    MoveL RelTool(pTarget,0,0,-2),vSpeed,z0,tTool\WObj:=wWobj;
    MoveL pTarget,vSpeed,fine,tTool\WObj:=wWobj;
    Set do_pen;
    MoveL pTarget,vSpeed,z0,tTool\WObj:=wWobj;
    MoveL pTarget,vSpeed,z0,tTool\WObj:=wWobj;
    MoveL pTarget,vSpeed,z0,tTool\WObj:=wWobj;
    MoveL pTarget,vSpeed,z0,tTool\WObj:=wWobj;
    MoveL pTarget,vSpeed,z0,tTool\WObj:=wWobj;
    MoveL pTarget,vSpeed,z0,tTool\WObj:=wWobj;
    MoveL pTarget,vSpeed,z0,tTool\WObj:=wWobj;
    MoveL pTarget,vSpeed,z0,tTool\WObj:=wWobj;
    MoveL pTarget,vSpeed,fine,tTool\WObj:=wWobj;
    Reset do_pen;
    MoveL RelTool(pTarget,0,0,-2),vSpeed,z0,tTool\WObj:=wWobj;
  ENDPROC
  PROC char_pipe()
    MoveL pTarget,vSpeed,fine,tTool\WObj:=wWobj;
    Set do_pen;
    MoveL pTarget,vSpeed,fine,tTool\WObj:=wWobj;
    Reset do_pen;
    MoveL RelTool(pTarget,0,0,-2),vSpeed,z0,tTool\WObj:=wWobj;
  ENDPROC
  PROC char_lessthan()
    MoveL pTarget,vSpeed,fine,tTool\WObj:=wWobj;
    Set do_pen;
    MoveL pTarget,vSpeed,z0,tTool\WObj:=wWobj;
    MoveL pTarget,vSpeed,fine,tTool\WObj:=wWobj;
    Reset do_pen;
    MoveL RelTool(pTarget,0,0,-2),vSpeed,z0,tTool\WObj:=wWobj;
  ENDPROC
  PROC char_greaterthan()
    MoveL pTarget,vSpeed,fine,tTool\WObj:=wWobj;
    Set do_pen;
    MoveL pTarget,vSpeed,z0,tTool\WObj:=wWobj;
    MoveL pTarget,vSpeed,fine,tTool\WObj:=wWobj;
    Reset do_pen;
    MoveL RelTool(pTarget,0,0,-2),vSpeed,z0,tTool\WObj:=wWobj;
  ENDPROC
  PROC char_question()
    MoveL pTarget,vSpeed,fine,tTool\WObj:=wWobj;
    Set do_pen;
    MoveL pTarget,vSpeed,z0,tTool\WObj:=wWobj;
    MoveL pTarget,vSpeed,z0,tTool\WObj:=wWobj;
    MoveL pTarget,vSpeed,z0,tTool\WObj:=wWobj;
    MoveL pTarget,vSpeed,z0,tTool\WObj:=wWobj;
    MoveL pTarget,vSpeed,z0,tTool\WObj:=wWobj;
    MoveL pTarget,vSpeed,z0,tTool\WObj:=wWobj;
    MoveL pTarget,vSpeed,z0,tTool\WObj:=wWobj;
    MoveL pTarget,vSpeed,z0,tTool\WObj:=wWobj;
    MoveL pTarget,vSpeed,z0,tTool\WObj:=wWobj;
    MoveL pTarget,vSpeed,z0,tTool\WObj:=wWobj;
    MoveL pTarget,vSpeed,z0,tTool\WObj:=wWobj;
    MoveL pTarget,vSpeed,z0,tTool\WObj:=wWobj;
    MoveL pTarget,vSpeed,fine,tTool\WObj:=wWobj;
    Reset do_pen;
    MoveL RelTool(pTarget,0,0,-2),vSpeed,z0,tTool\WObj:=wWobj;
    MoveL pTarget,vSpeed,fine,tTool\WObj:=wWobj;
    Set do_pen;
    MoveL pTarget,vSpeed,z0,tTool\WObj:=wWobj;
    MoveL pTarget,vSpeed,z0,tTool\WObj:=wWobj;
    MoveL pTarget,vSpeed,z0,tTool\WObj:=wWobj;
    MoveL pTarget,vSpeed,fine,tTool\WObj:=wWobj;
    Reset do_pen;
    MoveL RelTool(pTarget,0,0,-2),vSpeed,z0,tTool\WObj:=wWobj;
  ENDPROC
  PROC char_underscore()
    MoveL pTarget,vSpeed,fine,tTool\WObj:=wWobj;
    Set do_pen;
    MoveL pTarget,vSpeed,fine,tTool\WObj:=wWobj;
    Reset do_pen;
    MoveL RelTool(pTarget,0,0,-2),vSpeed,z0,tTool\WObj:=wWobj;
  ENDPROC
  PROC char_minus()
    MoveL pTarget,vSpeed,fine,tTool\WObj:=wWobj;
    Set do_pen;
    MoveL pTarget,vSpeed,fine,tTool\WObj:=wWobj;
    Reset do_pen;
    MoveL RelTool(pTarget,0,0,-2),vSpeed,z0,tTool\WObj:=wWobj;
  ENDPROC
  PROC char_tilde()
    MoveL pTarget,vSpeed,fine,tTool\WObj:=wWobj;
    Set do_pen;
    MoveL pTarget,vSpeed,z0,tTool\WObj:=wWobj;
    MoveL pTarget,vSpeed,z0,tTool\WObj:=wWobj;
    MoveL pTarget,vSpeed,z0,tTool\WObj:=wWobj;
    MoveL pTarget,vSpeed,z0,tTool\WObj:=wWobj;
    MoveL pTarget,vSpeed,z0,tTool\WObj:=wWobj;
    MoveL pTarget,vSpeed,z0,tTool\WObj:=wWobj;
    MoveL pTarget,vSpeed,z0,tTool\WObj:=wWobj;
    MoveL pTarget,vSpeed,z0,tTool\WObj:=wWobj;
    MoveL pTarget,vSpeed,z0,tTool\WObj:=wWobj;
    MoveL pTarget,vSpeed,fine,tTool\WObj:=wWobj;
    Reset do_pen;
    MoveL RelTool(pTarget,0,0,-2),vSpeed,z0,tTool\WObj:=wWobj;
    MoveL pTarget,vSpeed,fine,tTool\WObj:=wWobj;
    Set do_pen;
    MoveL pTarget,vSpeed,z0,tTool\WObj:=wWobj;
    MoveL pTarget,vSpeed,z0,tTool\WObj:=wWobj;
    MoveL pTarget,vSpeed,z0,tTool\WObj:=wWobj;
    MoveL pTarget,vSpeed,z0,tTool\WObj:=wWobj;
    MoveL pTarget,vSpeed,z0,tTool\WObj:=wWobj;
    MoveL pTarget,vSpeed,z0,tTool\WObj:=wWobj;
    MoveL pTarget,vSpeed,z0,tTool\WObj:=wWobj;
    MoveL pTarget,vSpeed,z0,tTool\WObj:=wWobj;
    MoveL pTarget,vSpeed,z0,tTool\WObj:=wWobj;
    MoveL pTarget,vSpeed,fine,tTool\WObj:=wWobj;
    Reset do_pen;
    MoveL RelTool(pTarget,0,0,-2),vSpeed,z0,tTool\WObj:=wWobj;
  ENDPROC
  PROC char_period()
    MoveL pTarget,vSpeed,fine,tTool\WObj:=wWobj;
    Set do_pen;
    MoveL pTarget,vSpeed,z0,tTool\WObj:=wWobj;
    MoveL pTarget,vSpeed,z0,tTool\WObj:=wWobj;
    MoveL pTarget,vSpeed,z0,tTool\WObj:=wWobj;
    MoveL pTarget,vSpeed,fine,tTool\WObj:=wWobj;
    Reset do_pen;
    MoveL RelTool(pTarget,0,0,-2),vSpeed,z0,tTool\WObj:=wWobj;
  ENDPROC
  PROC char_comma()
    MoveL pTarget,vSpeed,fine,tTool\WObj:=wWobj;
    Set do_pen;
    MoveL pTarget,vSpeed,z0,tTool\WObj:=wWobj;
    MoveL pTarget,vSpeed,z0,tTool\WObj:=wWobj;
    MoveL pTarget,vSpeed,z0,tTool\WObj:=wWobj;
    MoveL pTarget,vSpeed,z0,tTool\WObj:=wWobj;
    MoveL pTarget,vSpeed,z0,tTool\WObj:=wWobj;
    MoveL pTarget,vSpeed,fine,tTool\WObj:=wWobj;
    Reset do_pen;
    MoveL RelTool(pTarget,0,0,-2),vSpeed,z0,tTool\WObj:=wWobj;
  ENDPROC
  PROC char_semicolon()
    MoveL pTarget,vSpeed,fine,tTool\WObj:=wWobj;
    Set do_pen;
    MoveL pTarget,vSpeed,z0,tTool\WObj:=wWobj;
    MoveL pTarget,vSpeed,z0,tTool\WObj:=wWobj;
    MoveL pTarget,vSpeed,z0,tTool\WObj:=wWobj;
    MoveL pTarget,vSpeed,fine,tTool\WObj:=wWobj;
    Reset do_pen;
    MoveL RelTool(pTarget,0,0,-2),vSpeed,z0,tTool\WObj:=wWobj;
    MoveL pTarget,vSpeed,fine,tTool\WObj:=wWobj;
    Set do_pen;
    MoveL pTarget,vSpeed,z0,tTool\WObj:=wWobj;
    MoveL pTarget,vSpeed,z0,tTool\WObj:=wWobj;
    MoveL pTarget,vSpeed,z0,tTool\WObj:=wWobj;
    MoveL pTarget,vSpeed,z0,tTool\WObj:=wWobj;
    MoveL pTarget,vSpeed,z0,tTool\WObj:=wWobj;
    MoveL pTarget,vSpeed,fine,tTool\WObj:=wWobj;
    Reset do_pen;
    MoveL RelTool(pTarget,0,0,-2),vSpeed,z0,tTool\WObj:=wWobj;
  ENDPROC
  PROC char_colon()
    MoveL pTarget,vSpeed,fine,tTool\WObj:=wWobj;
    Set do_pen;
    MoveL pTarget,vSpeed,z0,tTool\WObj:=wWobj;
    MoveL pTarget,vSpeed,z0,tTool\WObj:=wWobj;
    MoveL pTarget,vSpeed,z0,tTool\WObj:=wWobj;
    MoveL pTarget,vSpeed,fine,tTool\WObj:=wWobj;
    Reset do_pen;
    MoveL RelTool(pTarget,0,0,-2),vSpeed,z0,tTool\WObj:=wWobj;
    MoveL pTarget,vSpeed,fine,tTool\WObj:=wWobj;
    Set do_pen;
    MoveL pTarget,vSpeed,z0,tTool\WObj:=wWobj;
    MoveL pTarget,vSpeed,z0,tTool\WObj:=wWobj;
    MoveL pTarget,vSpeed,z0,tTool\WObj:=wWobj;
    MoveL pTarget,vSpeed,fine,tTool\WObj:=wWobj;
    Reset do_pen;
    MoveL RelTool(pTarget,0,0,-2),vSpeed,z0,tTool\WObj:=wWobj;
  ENDPROC
ENDMODULE


--- Controller Data/IRB1200_5_90/RAPID/TASK1/PROGMOD/hersheyCursiveModule.modx ---
MODULE hersheyCursiveModule
    ! Character: a
    PROC char_a(\num nScaleParam)
        VAR robtarget pTarget;
        VAR num nScale:=1;
        pTarget:=refTarget;
        IF Present(nScaleParam) THEN
            nScale:=nScaleParam;
        ENDIF
        pTarget.trans:=[9*nScale,17.0*nScale,0];
        MoveL pTarget,vSpeed,fine,tTool\WObj:=wWobj;
        Set do_pen;
        pTarget.trans:=[8*nScale,19.0*nScale,0];
        MoveL pTarget,vSpeed,z0,tTool\WObj:=wWobj;
        pTarget.trans:=[6*nScale,20.0*nScale,0];
        MoveL pTarget,vSpeed,z0,tTool\WObj:=wWobj;
        pTarget.trans:=[4*nScale,20.0*nScale,0];
        MoveL pTarget,vSpeed,z0,tTool\WObj:=wWobj;
        pTarget.trans:=[2*nScale,19.0*nScale,0];
        MoveL pTarget,vSpeed,z0,tTool\WObj:=wWobj;
        pTarget.trans:=[1*nScale,18.0*nScale,0];
        MoveL pTarget,vSpeed,z0,tTool\WObj:=wWobj;
        pTarget.trans:=[0*nScale,16.0*nScale,0];
        MoveL pTarget,vSpeed,z0,tTool\WObj:=wWobj;
        pTarget.trans:=[0*nScale,14.0*nScale,0];
        MoveL pTarget,vSpeed,z0,tTool\WObj:=wWobj;
        pTarget.trans:=[1*nScale,12.0*nScale,0];
        MoveL pTarget,vSpeed,z0,tTool\WObj:=wWobj;
        pTarget.trans:=[3*nScale,11.0*nScale,0];
        MoveL pTarget,vSpeed,z0,tTool\WObj:=wWobj;
        pTarget.trans:=[5*nScale,11.0*nScale,0];
        MoveL pTarget,vSpeed,z0,tTool\WObj:=wWobj;
        pTarget.trans:=[7*nScale,12.0*nScale,0];
        MoveL pTarget,vSpeed,z0,tTool\WObj:=wWobj;
        pTarget.trans:=[8*nScale,14.0*nScale,0];
        MoveL pTarget,vSpeed,z0,tTool\WObj:=wWobj;
        pTarget.trans:=[10*nScale,20.0*nScale,0];
        MoveL pTarget,vSpeed,z0,tTool\WObj:=wWobj;
        pTarget.trans:=[9*nScale,15.0*nScale,0];
        MoveL pTarget,vSpeed,z0,tTool\WObj:=wWobj;
        pTarget.trans:=[9*nScale,12.0*nScale,0];
        MoveL pTarget,vSpeed,z0,tTool\WObj:=wWobj;
        pTarget.trans:=[10*nScale,11.0*nScale,0];
        MoveL pTarget,vSpeed,z0,tTool\WObj:=wWobj;
        pTarget.trans:=[11*nScale,11.0*nScale,0];
        MoveL pTarget,vSpeed,z0,tTool\WObj:=wWobj;
        pTarget.trans:=[13*nScale,12.0*nScale,0];
        MoveL pTarget,vSpeed,z0,tTool\WObj:=wWobj;
        pTarget.trans:=[14*nScale,13.0*nScale,0];
        MoveL pTarget,vSpeed,z0,tTool\WObj:=wWobj;
        pTarget.trans:=[16*nScale,16.0*nScale,0];
        MoveL pTarget,vSpeed,fine,tTool\WObj:=wWobj;
        Reset do_pen;
        MoveL RelTool(pTarget,0,0,-2),vSpeed,z0,tTool\WObj:=wWobj;
        wWobj.oframe.trans.x:=wWobj.oframe.trans.x+16*nScale;
    ENDPROC

    ! Character: b
    PROC char_b(\num nScaleParam)
        VAR robtarget pTarget;
        VAR num nScale:=1;
        pTarget:=refTarget;
        IF Present(nScaleParam) THEN
            nScale:=nScaleParam;
        ENDIF
        pTarget.trans:=[0*nScale,16.0*nScale,0];
        MoveL pTarget,vSpeed,fine,tTool\WObj:=wWobj;
        Set do_pen;
        pTarget.trans:=[2*nScale,19.0*nScale,0];
        MoveL pTarget,vSpeed,z0,tTool\WObj:=wWobj;
        pTarget.trans:=[5*nScale,24.0*nScale,0];
        MoveL pTarget,vSpeed,z0,tTool\WObj:=wWobj;
        pTarget.trans:=[6*nScale,26.0*nScale,0];
        MoveL pTarget,vSpeed,z0,tTool\WObj:=wWobj;
        pTarget.trans:=[7*nScale,29.0*nScale,0];
        MoveL pTarget,vSpeed,z0,tTool\WObj:=wWobj;
        pTarget.trans:=[7*nScale,31.0*nScale,0];
        MoveL pTarget,vSpeed,z0,tTool\WObj:=wWobj;
        pTarget.trans:=[6*nScale,32.0*nScale,0];
        MoveL pTarget,vSpeed,z0,tTool\WObj:=wWobj;
        pTarget.trans:=[4*nScale,31.0*nScale,0];
        MoveL pTarget,vSpeed,z0,tTool\WObj:=wWobj;
        pTarget.trans:=[3*nScale,29.0*nScale,0];
        MoveL pTarget,vSpeed,z0,tTool\WObj:=wWobj;
        pTarget.trans:=[2*nScale,25.0*nScale,0];
        MoveL pTarget,vSpeed,z0,tTool\WObj:=wWobj;
        pTarget.trans:=[1*nScale,18.0*nScale,0];
        MoveL pTarget,vSpeed,z0,tTool\WObj:=wWobj;
        pTarget.trans:=[1*nScale,12.0*nScale,0];
        MoveL pTarget,vSpeed,z0,tTool\WObj:=wWobj;
        pTarget.trans:=[2*nScale,11.0*nScale,0];
        MoveL pTarget,vSpeed,z0,tTool\WObj:=wWobj;
        pTarget.trans:=[3*nScale,11.0*nScale,0];
        MoveL pTarget,vSpeed,z0,tTool\WObj:=wWobj;
        pTarget.trans:=[5*nScale,12.0*nScale,0];
        MoveL pTarget,vSpeed,z0,tTool\WObj:=wWobj;
        pTarget.trans:=[7*nScale,14.0*nScale,0];
        MoveL pTarget,vSpeed,z0,tTool\WObj:=wWobj;
        pTarget.trans:=[8*nScale,17.0*nScale,0];
        MoveL pTarget,vSpeed,z0,tTool\WObj:=wWobj;
        pTarget.trans:=[8*nScale,20.0*nScale,0];
        MoveL pTarget,vSpeed,z0,tTool\WObj:=wWobj;
        pTarget.trans:=[9*nScale,16.0*nScale,0];
        MoveL pTarget,vSpeed,z0,tTool\WObj:=wWobj;
        pTarget.trans:=[10*nScale,15.0*nScale,0];
        MoveL pTarget,vSpeed,z0,tTool\WObj:=wWobj;
        pTarget.trans:=[12*nScale,15.0*nScale,0];
        MoveL pTarget,vSpeed,z0,tTool\WObj:=wWobj;
        pTarget.trans:=[14*nScale,16.0*nScale,0];
        MoveL pTarget,vSpeed,fine,tTool\WObj:=wWobj;
        Reset do_pen;
        MoveL RelTool(pTarget,0,0,-2),vSpeed,z0,tTool\WObj:=wWobj;
        wWobj.oframe.trans.x:=wWobj.oframe.trans.x+14*nScale;
    ENDPROC

    ! Character: c
    PROC char_c(\num nScaleParam)
        VAR robtarget pTarget;
        VAR num nScale:=1;
        pTarget:=refTarget;
        IF Present(nScaleParam) THEN
            nScale:=nScaleParam;
        ENDIF
        pTarget.trans:=[7*nScale,18.0*nScale,0];
        MoveL pTarget,vSpeed,fine,tTool\WObj:=wWobj;
        Set do_pen;
        pTarget.trans:=[7*nScale,19.0*nScale,0];
        MoveL pTarget,vSpeed,z0,tTool\WObj:=wWobj;
        pTarget.trans:=[6*nScale,20.0*nScale,0];
        MoveL pTarget,vSpeed,z0,tTool\WObj:=wWobj;
        pTarget.trans:=[4*nScale,20.0*nScale,0];
        MoveL pTarget,vSpeed,z0,tTool\WObj:=wWobj;
        pTarget.trans:=[2*nScale,19.0*nScale,0];
        MoveL pTarget,vSpeed,z0,tTool\WObj:=wWobj;
        pTarget.trans:=[1*nScale,18.0*nScale,0];
        MoveL pTarget,vSpeed,z0,tTool\WObj:=wWobj;
        pTarget.trans:=[0*nScale,16.0*nScale,0];
        MoveL pTarget,vSpeed,z0,tTool\WObj:=wWobj;
        pTarget.trans:=[0*nScale,14.0*nScale,0];
        MoveL pTarget,vSpeed,z0,tTool\WObj:=wWobj;
        pTarget.trans:=[1*nScale,12.0*nScale,0];
        MoveL pTarget,vSpeed,z0,tTool\WObj:=wWobj;
        pTarget.trans:=[3*nScale,11.0*nScale,0];
        MoveL pTarget,vSpeed,z0,tTool\WObj:=wWobj;
        pTarget.trans:=[6*nScale,11.0*nScale,0];
        MoveL pTarget,vSpeed,z0,tTool\WObj:=wWobj;
        pTarget.trans:=[9*nScale,13.0*nScale,0];
        MoveL pTarget,vSpeed,z0,tTool\WObj:=wWobj;
        pTarget.trans:=[11*nScale,16.0*nScale,0];
        MoveL pTarget,vSpeed,fine,tTool\WObj:=wWobj;
        Reset do_pen;
        MoveL RelTool(pTarget,0,0,-2),vSpeed,z0,tTool\WObj:=wWobj;
        wWobj.oframe.trans.x:=wWobj.oframe.trans.x+11*nScale;
    ENDPROC

    ! Character: d
    PROC char_d(\num nScaleParam)
        VAR robtarget pTarget;
        VAR num nScale:=1;
        pTarget:=refTarget;
        IF Present(nScaleParam) THEN
            nScale:=nScaleParam;
        ENDIF
        pTarget.trans:=[9*nScale,17.0*nScale,0];
        MoveL pTarget,vSpeed,fine,tTool\WObj:=wWobj;
        Set do_pen;
        pTarget.trans:=[8*nScale,19.0*nScale,0];
        MoveL pTarget,vSpeed,z0,tTool\WObj:=wWobj;
        pTarget.trans:=[6*nScale,20.0*nScale,0];
        MoveL pTarget,vSpeed,z0,tTool\WObj:=wWobj;
        pTarget.trans:=[4*nScale,20.0*nScale,0];
        MoveL pTarget,vSpeed,z0,tTool\WObj:=wWobj;
        pTarget.trans:=[2*nScale,19.0*nScale,0];
        MoveL pTarget,vSpeed,z0,tTool\WObj:=wWobj;
        pTarget.trans:=[1*nScale,18.0*nScale,0];
        MoveL pTarget,vSpeed,z0,tTool\WObj:=wWobj;
        pTarget.trans:=[0*nScale,16.0*nScale,0];
        MoveL pTarget,vSpeed,z0,tTool\WObj:=wWobj;
        pTarget.trans:=[0*nScale,14.0*nScale,0];
        MoveL pTarget,vSpeed,z0,tTool\WObj:=wWobj;
        pTarget.trans:=[1*nScale,12.0*nScale,0];
        MoveL pTarget,vSpeed,z0,tTool\WObj:=wWobj;
        pTarget.trans:=[3*nScale,11.0*nScale,0];
        MoveL pTarget,vSpeed,z0,tTool\WObj:=wWobj;
        pTarget.trans:=[5*nScale,11.0*nScale,0];
        MoveL pTarget,vSpeed,z0,tTool\WObj:=wWobj;
        pTarget.trans:=[7*nScale,12.0*nScale,0];
        MoveL pTarget,vSpeed,z0,tTool\WObj:=wWobj;
        pTarget.trans:=[8*nScale,14.0*nScale,0];
        MoveL pTarget,vSpeed,z0,tTool\WObj:=wWobj;
        pTarget.trans:=[14*nScale,32.0*nScale,0];
        MoveL pTarget,vSpeed,fine,tTool\WObj:=wWobj;
        Reset do_pen;
        MoveL RelTool(pTarget,0,0,-2),vSpeed,z0,tTool\WObj:=wWobj;
        pTarget.trans:=[10*nScale,20.0*nScale,0];
        MoveL pTarget,vSpeed,fine,tTool\WObj:=wWobj;
        Set do_pen;
        pTarget.trans:=[9*nScale,15.0*nScale,0];
        MoveL pTarget,vSpeed,z0,tTool\WObj:=wWobj;
        pTarget.trans:=[9*nScale,12.0*nScale,0];
        MoveL pTarget,vSpeed,z0,tTool\WObj:=wWobj;
        pTarget.trans:=[10*nScale,11.0*nScale,0];
        MoveL pTarget,vSpeed,z0,tTool\WObj:=wWobj;
        pTarget.trans:=[11*nScale,11.0*nScale,0];
        MoveL pTarget,vSpeed,z0,tTool\WObj:=wWobj;
        pTarget.trans:=[13*nScale,12.0*nScale,0];
        MoveL pTarget,vSpeed,z0,tTool\WObj:=wWobj;
        pTarget.trans:=[14*nScale,13.0*nScale,0];
        MoveL pTarget,vSpeed,z0,tTool\WObj:=wWobj;
        pTarget.trans:=[16*nScale,16.0*nScale,0];
        MoveL pTarget,vSpeed,fine,tTool\WObj:=wWobj;
        Reset do_pen;
        MoveL RelTool(pTarget,0,0,-2),vSpeed,z0,tTool\WObj:=wWobj;
        wWobj.oframe.trans.x:=wWobj.oframe.trans.x+16*nScale;
    ENDPROC

    ! Character: e
    PROC char_e(\num nScaleParam)
        VAR robtarget pTarget;
        VAR num nScale:=1;
        pTarget:=refTarget;
        IF Present(nScaleParam) THEN
            nScale:=nScaleParam;
        ENDIF
        pTarget.trans:=[1*nScale,13.0*nScale,0];
        MoveL pTarget,vSpeed,fine,tTool\WObj:=wWobj;
        Set do_pen;
        pTarget.trans:=[3*nScale,14.0*nScale,0];
        MoveL pTarget,vSpeed,z0,tTool\WObj:=wWobj;
        pTarget.trans:=[4*nScale,15.0*nScale,0];
        MoveL pTarget,vSpeed,z0,tTool\WObj:=wWobj;
        pTarget.trans:=[5*nScale,17.0*nScale,0];
        MoveL pTarget,vSpeed,z0,tTool\WObj:=wWobj;
        pTarget.trans:=[5*nScale,19.0*nScale,0];
        MoveL pTarget,vSpeed,z0,tTool\WObj:=wWobj;
        pTarget.trans:=[4*nScale,20.0*nScale,0];
        MoveL pTarget,vSpeed,z0,tTool\WObj:=wWobj;
        pTarget.trans:=[3*nScale,20.0*nScale,0];
        MoveL pTarget,vSpeed,z0,tTool\WObj:=wWobj;
        pTarget.trans:=[1*nScale,19.0*nScale,0];
        MoveL pTarget,vSpeed,z0,tTool\WObj:=wWobj;
        pTarget.trans:=[0*nScale,17.0*nScale,0];
        MoveL pTarget,vSpeed,z0,tTool\WObj:=wWobj;
        pTarget.trans:=[0*nScale,14.0*nScale,0];
        MoveL pTarget,vSpeed,z0,tTool\WObj:=wWobj;
        pTarget.trans:=[1*nScale,12.0*nScale,0];
        MoveL pTarget,vSpeed,z0,tTool\WObj:=wWobj;
        pTarget.trans:=[3*nScale,11.0*nScale,0];
        MoveL pTarget,vSpeed,z0,tTool\WObj:=wWobj;
        pTarget.trans:=[5*nScale,11.0*nScale,0];
        MoveL pTarget,vSpeed,z0,tTool\WObj:=wWobj;
        pTarget.trans:=[7*nScale,12.0*nScale,0];
        MoveL pTarget,vSpeed,z0,tTool\WObj:=wWobj;
        pTarget.trans:=[8*nScale,13.0*nScale,0];
        MoveL pTarget,vSpeed,z0,tTool\WObj:=wWobj;
        pTarget.trans:=[10*nScale,16.0*nScale,0];
        MoveL pTarget,vSpeed,fine,tTool\WObj:=wWobj;
        Reset do_pen;
        MoveL RelTool(pTarget,0,0,-2),vSpeed,z0,tTool\WObj:=wWobj;
        wWobj.oframe.trans.x:=wWobj.oframe.trans.x+10*nScale;
    ENDPROC

    ! Character: f
    PROC char_f(\num nScaleParam)
        VAR robtarget pTarget;
        VAR num nScale:=1;
        pTarget:=refTarget;
        IF Present(nScaleParam) THEN
            nScale:=nScaleParam;
        ENDIF
        pTarget.trans:=[0*nScale,16.0*nScale,0];
        MoveL pTarget,vSpeed,fine,tTool\WObj:=wWobj;
        Set do_pen;
        pTarget.trans:=[4*nScale,21.0*nScale,0];
        MoveL pTarget,vSpeed,z0,tTool\WObj:=wWobj;
        pTarget.trans:=[6*nScale,24.0*nScale,0];
        MoveL pTarget,vSpeed,z0,tTool\WObj:=wWobj;
        pTarget.trans:=[7*nScale,26.0*nScale,0];
        MoveL pTarget,vSpeed,z0,tTool\WObj:=wWobj;
        pTarget.trans:=[8*nScale,29.0*nScale,0];
        MoveL pTarget,vSpeed,z0,tTool\WObj:=wWobj;
        pTarget.trans:=[8*nScale,31.0*nScale,0];
        MoveL pTarget,vSpeed,z0,tTool\WObj:=wWobj;
        pTarget.trans:=[7*nScale,32.0*nScale,0];
        MoveL pTarget,vSpeed,z0,tTool\WObj:=wWobj;
        pTarget.trans:=[5*nScale,31.0*nScale,0];
        MoveL pTarget,vSpeed,z0,tTool\WObj:=wWobj;
        pTarget.trans:=[4*nScale,29.0*nScale,0];
        MoveL pTarget,vSpeed,z0,tTool\WObj:=wWobj;
        pTarget.trans:=[2*nScale,21.0*nScale,0];
        MoveL pTarget,vSpeed,z0,tTool\WObj:=wWobj;
        pTarget.trans:=[-1*nScale,12.0*nScale,0];
        MoveL pTarget,vSpeed,z0,tTool\WObj:=wWobj;
        pTarget.trans:=[-4*nScale,5.0*nScale,0];
        MoveL pTarget,vSpeed,z0,tTool\WObj:=wWobj;
        pTarget.trans:=[-5*nScale,2.0*nScale,0];
        MoveL pTarget,vSpeed,z0,tTool\WObj:=wWobj;
        pTarget.trans:=[-5*nScale,0.0*nScale,0];
        MoveL pTarget,vSpeed,z0,tTool\WObj:=wWobj;
        pTarget.trans:=[-4*nScale,-1.0*nScale,0];
        MoveL pTarget,vSpeed,z0,tTool\WObj:=wWobj;
        pTarget.trans:=[-2*nScale,0.0*nScale,0];
        MoveL pTarget,vSpeed,z0,tTool\WObj:=wWobj;
        pTarget.trans:=[-1*nScale,3.0*nScale,0];
        MoveL pTarget,vSpeed,z0,tTool\WObj:=wWobj;
        pTarget.trans:=[0*nScale,12.0*nScale,0];
        MoveL pTarget,vSpeed,z0,tTool\WObj:=wWobj;
        pTarget.trans:=[1*nScale,11.0*nScale,0];
        MoveL pTarget,vSpeed,z0,tTool\WObj:=wWobj;
        pTarget.trans:=[3*nScale,11.0*nScale,0];
        MoveL pTarget,vSpeed,z0,tTool\WObj:=wWobj;
        pTarget.trans:=[5*nScale,12.0*nScale,0];
        MoveL pTarget,vSpeed,z0,tTool\WObj:=wWobj;
        pTarget.trans:=[6*nScale,13.0*nScale,0];
        MoveL pTarget,vSpeed,z0,tTool\WObj:=wWobj;
        pTarget.trans:=[8*nScale,16.0*nScale,0];
        MoveL pTarget,vSpeed,fine,tTool\WObj:=wWobj;
        Reset do_pen;
        MoveL RelTool(pTarget,0,0,-2),vSpeed,z0,tTool\WObj:=wWobj;
        wWobj.oframe.trans.x:=wWobj.oframe.trans.x+8*nScale;
    ENDPROC

    ! Character: g
    PROC char_g(\num nScaleParam)
        VAR robtarget pTarget;
        VAR num nScale:=1;
        pTarget:=refTarget;
        IF Present(nScaleParam) THEN
            nScale:=nScaleParam;
        ENDIF
        pTarget.trans:=[9*nScale,17.0*nScale,0];
        MoveL pTarget,vSpeed,fine,tTool\WObj:=wWobj;
        Set do_pen;
        pTarget.trans:=[8*nScale,19.0*nScale,0];
        MoveL pTarget,vSpeed,z0,tTool\WObj:=wWobj;
        pTarget.trans:=[6*nScale,20.0*nScale,0];
        MoveL pTarget,vSpeed,z0,tTool\WObj:=wWobj;
        pTarget.trans:=[4*nScale,20.0*nScale,0];
        MoveL pTarget,vSpeed,z0,tTool\WObj:=wWobj;
        pTarget.trans:=[2*nScale,19.0*nScale,0];
        MoveL pTarget,vSpeed,z0,tTool\WObj:=wWobj;
        pTarget.trans:=[1*nScale,18.0*nScale,0];
        MoveL pTarget,vSpeed,z0,tTool\WObj:=wWobj;
        pTarget.trans:=[0*nScale,16.0*nScale,0];
        MoveL pTarget,vSpeed,z0,tTool\WObj:=wWobj;
        pTarget.trans:=[0*nScale,14.0*nScale,0];
        MoveL pTarget,vSpeed,z0,tTool\WObj:=wWobj;
        pTarget.trans:=[1*nScale,12.0*nScale,0];
        MoveL pTarget,vSpeed,z0,tTool\WObj:=wWobj;
        pTarget.trans:=[3*nScale,11.0*nScale,0];
        MoveL pTarget,vSpeed,z0,tTool\WObj:=wWobj;
        pTarget.trans:=[5*nScale,11.0*nScale,0];
        MoveL pTarget,vSpeed,z0,tTool\WObj:=wWobj;
        pTarget.trans:=[7*nScale,12.0*nScale,0];
        MoveL pTarget,vSpeed,z0,tTool\WObj:=wWobj;
        pTarget.trans:=[8*nScale,13.0*nScale,0];
        MoveL pTarget,vSpeed,fine,tTool\WObj:=wWobj;
        Reset do_pen;
        MoveL RelTool(pTarget,0,0,-2),vSpeed,z0,tTool\WObj:=wWobj;
        pTarget.trans:=[10*nScale,20.0*nScale,0];
        MoveL pTarget,vSpeed,fine,tTool\WObj:=wWobj;
        Set do_pen;
        pTarget.trans:=[8*nScale,13.0*nScale,0];
        MoveL pTarget,vSpeed,z0,tTool\WObj:=wWobj;
        pTarget.trans:=[4*nScale,2.0*nScale,0];
        MoveL pTarget,vSpeed,z0,tTool\WObj:=wWobj;
        pTarget.trans:=[3*nScale,0.0*nScale,0];
        MoveL pTarget,vSpeed,z0,tTool\WObj:=wWobj;
        pTarget.trans:=[1*nScale,-1.0*nScale,0];
        MoveL pTarget,vSpeed,z0,tTool\WObj:=wWobj;
        pTarget.trans:=[0*nScale,0.0*nScale,0];
        MoveL pTarget,vSpeed,z0,tTool\WObj:=wWobj;
        pTarget.trans:=[0*nScale,2.0*nScale,0];
        MoveL pTarget,vSpeed,z0,tTool\WObj:=wWobj;
        pTarget.trans:=[1*nScale,5.0*nScale,0];
        MoveL pTarget,vSpeed,z0,tTool\WObj:=wWobj;
        pTarget.trans:=[4*nScale,8.0*nScale,0];
        MoveL pTarget,vSpeed,z0,tTool\WObj:=wWobj;
        pTarget.trans:=[7*nScale,10.0*nScale,0];
        MoveL pTarget,vSpeed,z0,tTool\WObj:=wWobj;
        pTarget.trans:=[9*nScale,11.0*nScale,0];
        MoveL pTarget,vSpeed,z0,tTool\WObj:=wWobj;
        pTarget.trans:=[12*nScale,13.0*nScale,0];
        MoveL pTarget,vSpeed,z0,tTool\WObj:=wWobj;
        pTarget.trans:=[15*nScale,16.0*nScale,0];
        MoveL pTarget,vSpeed,fine,tTool\WObj:=wWobj;
        Reset do_pen;
        MoveL RelTool(pTarget,0,0,-2),vSpeed,z0,tTool\WObj:=wWobj;
        wWobj.oframe.trans.x:=wWobj.oframe.trans.x+15*nScale;
    ENDPROC

    ! Character: h
    PROC char_h(\num nScaleParam)
        VAR robtarget pTarget;
        VAR num nScale:=1;
        pTarget:=refTarget;
        IF Present(nScaleParam) THEN
            nScale:=nScaleParam;
        ENDIF
        pTarget.trans:=[0*nScale,16.0*nScale,0];
        MoveL pTarget,vSpeed,fine,tTool\WObj:=wWobj;
        Set do_pen;
        pTarget.trans:=[2*nScale,19.0*nScale,0];
        MoveL pTarget,vSpeed,z0,tTool\WObj:=wWobj;
        pTarget.trans:=[5*nScale,24.0*nScale,0];
        MoveL pTarget,vSpeed,z0,tTool\WObj:=wWobj;
        pTarget.trans:=[6*nScale,26.0*nScale,0];
        MoveL pTarget,vSpeed,z0,tTool\WObj:=wWobj;
        pTarget.trans:=[7*nScale,29.0*nScale,0];
        MoveL pTarget,vSpeed,z0,tTool\WObj:=wWobj;
        pTarget.trans:=[7*nScale,31.0*nScale,0];
        MoveL pTarget,vSpeed,z0,tTool\WObj:=wWobj;
        pTarget.trans:=[6*nScale,32.0*nScale,0];
        MoveL pTarget,vSpeed,z0,tTool\WObj:=wWobj;
        pTarget.trans:=[4*nScale,31.0*nScale,0];
        MoveL pTarget,vSpeed,z0,tTool\WObj:=wWobj;
        pTarget.trans:=[3*nScale,29.0*nScale,0];
        MoveL pTarget,vSpeed,z0,tTool\WObj:=wWobj;
        pTarget.trans:=[2*nScale,25.0*nScale,0];
        MoveL pTarget,vSpeed,z0,tTool\WObj:=wWobj;
        pTarget.trans:=[1*nScale,19.0*nScale,0];
        MoveL pTarget,vSpeed,z0,tTool\WObj:=wWobj;
        pTarget.trans:=[0*nScale,11.0*nScale,0];
        MoveL pTarget,vSpeed,fine,tTool\WObj:=wWobj;
        Reset do_pen;
        MoveL RelTool(pTarget,0,0,-2),vSpeed,z0,tTool\WObj:=wWobj;
        pTarget.trans:=[0*nScale,11.0*nScale,0];
        MoveL pTarget,vSpeed,fine,tTool\WObj:=wWobj;
        Set do_pen;
        pTarget.trans:=[1*nScale,14.0*nScale,0];
        MoveL pTarget,vSpeed,z0,tTool\WObj:=wWobj;
        pTarget.trans:=[2*nScale,16.0*nScale,0];
        MoveL pTarget,vSpeed,z0,tTool\WObj:=wWobj;
        pTarget.trans:=[4*nScale,19.0*nScale,0];
        MoveL pTarget,vSpeed,z0,tTool\WObj:=wWobj;
        pTarget.trans:=[6*nScale,20.0*nScale,0];
        MoveL pTarget,vSpeed,z0,tTool\WObj:=wWobj;
        pTarget.trans:=[8*nScale,20.0*nScale,0];
        MoveL pTarget,vSpeed,z0,tTool\WObj:=wWobj;
        pTarget.trans:=[9*nScale,19.0*nScale,0];
        MoveL pTarget,vSpeed,z0,tTool\WObj:=wWobj;
        pTarget.trans:=[9*nScale,17.0*nScale,0];
        MoveL pTarget,vSpeed,z0,tTool\WObj:=wWobj;
        pTarget.trans:=[8*nScale,14.0*nScale,0];
        MoveL pTarget,vSpeed,z0,tTool\WObj:=wWobj;
        pTarget.trans:=[8*nScale,12.0*nScale,0];
        MoveL pTarget,vSpeed,z0,tTool\WObj:=wWobj;
        pTarget.trans:=[9*nScale,11.0*nScale,0];
        MoveL pTarget,vSpeed,z0,tTool\WObj:=wWobj;
        pTarget.trans:=[10*nScale,11.0*nScale,0];
        MoveL pTarget,vSpeed,z0,tTool\WObj:=wWobj;
        pTarget.trans:=[12*nScale,12.0*nScale,0];
        MoveL pTarget,vSpeed,z0,tTool\WObj:=wWobj;
        pTarget.trans:=[13*nScale,13.0*nScale,0];
        MoveL pTarget,vSpeed,z0,tTool\WObj:=wWobj;
        pTarget.trans:=[15*nScale,16.0*nScale,0];
        MoveL pTarget,vSpeed,fine,tTool\WObj:=wWobj;
        Reset do_pen;
        MoveL RelTool(pTarget,0,0,-2),vSpeed,z0,tTool\WObj:=wWobj;
        wWobj.oframe.trans.x:=wWobj.oframe.trans.x+15*nScale;
    ENDPROC

    ! Character: i
    PROC char_i(\num nScaleParam)
        VAR robtarget pTarget;
        VAR num nScale:=1;
        pTarget:=refTarget;
        IF Present(nScaleParam) THEN
            nScale:=nScaleParam;
        ENDIF
        pTarget.trans:=[3*nScale,25.0*nScale,0];
        MoveL pTarget,vSpeed,fine,tTool\WObj:=wWobj;
        Set do_pen;
        pTarget.trans:=[3*nScale,24.0*nScale,0];
        MoveL pTarget,vSpeed,z0,tTool\WObj:=wWobj;
        pTarget.trans:=[4*nScale,24.0*nScale,0];
        MoveL pTarget,vSpeed,z0,tTool\WObj:=wWobj;
        pTarget.trans:=[4*nScale,25.0*nScale,0];
        MoveL pTarget,vSpeed,z0,tTool\WObj:=wWobj;
        pTarget.trans:=[3*nScale,25.0*nScale,0];
        MoveL pTarget,vSpeed,fine,tTool\WObj:=wWobj;
        Reset do_pen;
        MoveL RelTool(pTarget,0,0,-2),vSpeed,z0,tTool\WObj:=wWobj;
        pTarget.trans:=[0*nScale,16.0*nScale,0];
        MoveL pTarget,vSpeed,fine,tTool\WObj:=wWobj;
        Set do_pen;
        pTarget.trans:=[2*nScale,20.0*nScale,0];
        MoveL pTarget,vSpeed,z0,tTool\WObj:=wWobj;
        pTarget.trans:=[0*nScale,14.0*nScale,0];
        MoveL pTarget,vSpeed,z0,tTool\WObj:=wWobj;
        pTarget.trans:=[0*nScale,12.0*nScale,0];
        MoveL pTarget,vSpeed,z0,tTool\WObj:=wWobj;
        pTarget.trans:=[1*nScale,11.0*nScale,0];
        MoveL pTarget,vSpeed,z0,tTool\WObj:=wWobj;
        pTarget.trans:=[2*nScale,11.0*nScale,0];
        MoveL pTarget,vSpeed,z0,tTool\WObj:=wWobj;
        pTarget.trans:=[4*nScale,12.0*nScale,0];
        MoveL pTarget,vSpeed,z0,tTool\WObj:=wWobj;
        pTarget.trans:=[5*nScale,13.0*nScale,0];
        MoveL pTarget,vSpeed,z0,tTool\WObj:=wWobj;
        pTarget.trans:=[7*nScale,16.0*nScale,0];
        MoveL pTarget,vSpeed,fine,tTool\WObj:=wWobj;
        Reset do_pen;
        MoveL RelTool(pTarget,0,0,-2),vSpeed,z0,tTool\WObj:=wWobj;
        wWobj.oframe.trans.x:=wWobj.oframe.trans.x+7*nScale;
    ENDPROC

    ! Character: j
    PROC char_j(\num nScaleParam)
        VAR robtarget pTarget;
        VAR num nScale:=1;
        pTarget:=refTarget;
        IF Present(nScaleParam) THEN
            nScale:=nScaleParam;
        ENDIF
        pTarget.trans:=[3*nScale,25.0*nScale,0];
        MoveL pTarget,vSpeed,fine,tTool\WObj:=wWobj;
        Set do_pen;
        pTarget.trans:=[3*nScale,24.0*nScale,0];
        MoveL pTarget,vSpeed,z0,tTool\WObj:=wWobj;
        pTarget.trans:=[4*nScale,24.0*nScale,0];
        MoveL pTarget,vSpeed,z0,tTool\WObj:=wWobj;
        pTarget.trans:=[4*nScale,25.0*nScale,0];
        MoveL pTarget,vSpeed,z0,tTool\WObj:=wWobj;
        pTarget.trans:=[3*nScale,25.0*nScale,0];
        MoveL pTarget,vSpeed,fine,tTool\WObj:=wWobj;
        Reset do_pen;
        MoveL RelTool(pTarget,0,0,-2),vSpeed,z0,tTool\WObj:=wWobj;
        pTarget.trans:=[0*nScale,16.0*nScale,0];
        MoveL pTarget,vSpeed,fine,tTool\WObj:=wWobj;
        Set do_pen;
        pTarget.trans:=[2*nScale,20.0*nScale,0];
        MoveL pTarget,vSpeed,z0,tTool\WObj:=wWobj;
        pTarget.trans:=[-4*nScale,2.0*nScale,0];
        MoveL pTarget,vSpeed,z0,tTool\WObj:=wWobj;
        pTarget.trans:=[-5*nScale,0.0*nScale,0];
        MoveL pTarget,vSpeed,z0,tTool\WObj:=wWobj;
        pTarget.trans:=[-7*nScale,-1.0*nScale,0];
        MoveL pTarget,vSpeed,z0,tTool\WObj:=wWobj;
        pTarget.trans:=[-8*nScale,0.0*nScale,0];
        MoveL pTarget,vSpeed,z0,tTool\WObj:=wWobj;
        pTarget.trans:=[-8*nScale,2.0*nScale,0];
        MoveL pTarget,vSpeed,z0,tTool\WObj:=wWobj;
        pTarget.trans:=[-7*nScale,5.0*nScale,0];
        MoveL pTarget,vSpeed,z0,tTool\WObj:=wWobj;
        pTarget.trans:=[-4*nScale,8.0*nScale,0];
        MoveL pTarget,vSpeed,z0,tTool\WObj:=wWobj;
        pTarget.trans:=[-1*nScale,10.0*nScale,0];
        MoveL pTarget,vSpeed,z0,tTool\WObj:=wWobj;
        pTarget.trans:=[1*nScale,11.0*nScale,0];
        MoveL pTarget,vSpeed,z0,tTool\WObj:=wWobj;
        pTarget.trans:=[4*nScale,13.0*nScale,0];
        MoveL pTarget,vSpeed,z0,tTool\WObj:=wWobj;
        pTarget.trans:=[7*nScale,16.0*nScale,0];
        MoveL pTarget,vSpeed,fine,tTool\WObj:=wWobj;
        Reset do_pen;
        MoveL RelTool(pTarget,0,0,-2),vSpeed,z0,tTool\WObj:=wWobj;
        wWobj.oframe.trans.x:=wWobj.oframe.trans.x+7*nScale;
    ENDPROC

    ! Character: k
    PROC char_k(\num nScaleParam)
        VAR robtarget pTarget;
        VAR num nScale:=1;
        pTarget:=refTarget;
        IF Present(nScaleParam) THEN
            nScale:=nScaleParam;
        ENDIF
        pTarget.trans:=[0*nScale,16.0*nScale,0];
        MoveL pTarget,vSpeed,fine,tTool\WObj:=wWobj;
        Set do_pen;
        pTarget.trans:=[2*nScale,19.0*nScale,0];
        MoveL pTarget,vSpeed,z0,tTool\WObj:=wWobj;
        pTarget.trans:=[5*nScale,24.0*nScale,0];
        MoveL pTarget,vSpeed,z0,tTool\WObj:=wWobj;
        pTarget.trans:=[6*nScale,26.0*nScale,0];
        MoveL pTarget,vSpeed,z0,tTool\WObj:=wWobj;
        pTarget.trans:=[7*nScale,29.0*nScale,0];
        MoveL pTarget,vSpeed,z0,tTool\WObj:=wWobj;
        pTarget.trans:=[7*nScale,31.0*nScale,0];
        MoveL pTarget,vSpeed,z0,tTool\WObj:=wWobj;
        pTarget.trans:=[6*nScale,32.0*nScale,0];
        MoveL pTarget,vSpeed,z0,tTool\WObj:=wWobj;
        pTarget.trans:=[4*nScale,31.0*nScale,0];
        MoveL pTarget,vSpeed,z0,tTool\WObj:=wWobj;
        pTarget.trans:=[3*nScale,29.0*nScale,0];
        MoveL pTarget,vSpeed,z0,tTool\WObj:=wWobj;
        pTarget.trans:=[2*nScale,25.0*nScale,0];
        MoveL pTarget,vSpeed,z0,tTool\WObj:=wWobj;
        pTarget.trans:=[1*nScale,19.0*nScale,0];
        MoveL pTarget,vSpeed,z0,tTool\WObj:=wWobj;
        pTarget.trans:=[0*nScale,11.0*nScale,0];
        MoveL pTarget,vSpeed,fine,tTool\WObj:=wWobj;
        Reset do_pen;
        MoveL RelTool(pTarget,0,0,-2),vSpeed,z0,tTool\WObj:=wWobj;
        pTarget.trans:=[0*nScale,11.0*nScale,0];
        MoveL pTarget,vSpeed,fine,tTool\WObj:=wWobj;
        Set do_pen;
        pTarget.trans:=[1*nScale,14.0*nScale,0];
        MoveL pTarget,vSpeed,z0,tTool\WObj:=wWobj;
        pTarget.trans:=[2*nScale,16.0*nScale,0];
        MoveL pTarget,vSpeed,z0,tTool\WObj:=wWobj;
        pTarget.trans:=[4*nScale,19.0*nScale,0];
        MoveL pTarget,vSpeed,z0,tTool\WObj:=wWobj;
        pTarget.trans:=[6*nScale,20.0*nScale,0];
        MoveL pTarget,vSpeed,z0,tTool\WObj:=wWobj;
        pTarget.trans:=[8*nScale,20.0*nScale,0];
        MoveL pTarget,vSpeed,z0,tTool\WObj:=wWobj;
        pTarget.trans:=[9*nScale,19.0*nScale,0];
        MoveL pTarget,vSpeed,z0,tTool\WObj:=wWobj;
        pTarget.trans:=[9*nScale,17.0*nScale,0];
        MoveL pTarget,vSpeed,z0,tTool\WObj:=wWobj;
        pTarget.trans:=[7*nScale,16.0*nScale,0];
        MoveL pTarget,vSpeed,z0,tTool\WObj:=wWobj;
        pTarget.trans:=[4*nScale,16.0*nScale,0];
        MoveL pTarget,vSpeed,fine,tTool\WObj:=wWobj;
        Reset do_pen;
        MoveL RelTool(pTarget,0,0,-2),vSpeed,z0,tTool\WObj:=wWobj;
        pTarget.trans:=[4*nScale,16.0*nScale,0];
        MoveL pTarget,vSpeed,fine,tTool\WObj:=wWobj;
        Set do_pen;
        pTarget.trans:=[6*nScale,15.0*nScale,0];
        MoveL pTarget,vSpeed,z0,tTool\WObj:=wWobj;
        pTarget.trans:=[7*nScale,12.0*nScale,0];
        MoveL pTarget,vSpeed,z0,tTool\WObj:=wWobj;
        pTarget.trans:=[8*nScale,11.0*nScale,0];
        MoveL pTarget,vSpeed,z0,tTool\WObj:=wWobj;
        pTarget.trans:=[9*nScale,11.0*nScale,0];
        MoveL pTarget,vSpeed,z0,tTool\WObj:=wWobj;
        pTarget.trans:=[11*nScale,12.0*nScale,0];
        MoveL pTarget,vSpeed,z0,tTool\WObj:=wWobj;
        pTarget.trans:=[12*nScale,13.0*nScale,0];
        MoveL pTarget,vSpeed,z0,tTool\WObj:=wWobj;
        pTarget.trans:=[14*nScale,16.0*nScale,0];
        MoveL pTarget,vSpeed,fine,tTool\WObj:=wWobj;
        Reset do_pen;
        MoveL RelTool(pTarget,0,0,-2),vSpeed,z0,tTool\WObj:=wWobj;
        wWobj.oframe.trans.x:=wWobj.oframe.trans.x+14*nScale;
    ENDPROC

    ! Character: l
    PROC char_l(\num nScaleParam)
        VAR robtarget pTarget;
        VAR num nScale:=1;
        pTarget:=refTarget;
        IF Present(nScaleParam) THEN
            nScale:=nScaleParam;
        ENDIF
        pTarget.trans:=[0*nScale,16.0*nScale,0];
        MoveL pTarget,vSpeed,fine,tTool\WObj:=wWobj;
        Set do_pen;
        pTarget.trans:=[2*nScale,19.0*nScale,0];
        MoveL pTarget,vSpeed,z0,tTool\WObj:=wWobj;
        pTarget.trans:=[5*nScale,24.0*nScale,0];
        MoveL pTarget,vSpeed,z0,tTool\WObj:=wWobj;
        pTarget.trans:=[6*nScale,26.0*nScale,0];
        MoveL pTarget,vSpeed,z0,tTool\WObj:=wWobj;
        pTarget.trans:=[7*nScale,29.0*nScale,0];
        MoveL pTarget,vSpeed,z0,tTool\WObj:=wWobj;
        pTarget.trans:=[7*nScale,31.0*nScale,0];
        MoveL pTarget,vSpeed,z0,tTool\WObj:=wWobj;
        pTarget.trans:=[6*nScale,32.0*nScale,0];
        MoveL pTarget,vSpeed,z0,tTool\WObj:=wWobj;
        pTarget.trans:=[4*nScale,31.0*nScale,0];
        MoveL pTarget,vSpeed,z0,tTool\WObj:=wWobj;
        pTarget.trans:=[3*nScale,29.0*nScale,0];
        MoveL pTarget,vSpeed,z0,tTool\WObj:=wWobj;
        pTarget.trans:=[2*nScale,25.0*nScale,0];
        MoveL pTarget,vSpeed,z0,tTool\WObj:=wWobj;
        pTarget.trans:=[1*nScale,18.0*nScale,0];
        MoveL pTarget,vSpeed,z0,tTool\WObj:=wWobj;
        pTarget.trans:=[1*nScale,12.0*nScale,0];
        MoveL pTarget,vSpeed,z0,tTool\WObj:=wWobj;
        pTarget.trans:=[2*nScale,11.0*nScale,0];
        MoveL pTarget,vSpeed,z0,tTool\WObj:=wWobj;
        pTarget.trans:=[3*nScale,11.0*nScale,0];
        MoveL pTarget,vSpeed,z0,tTool\WObj:=wWobj;
        pTarget.trans:=[5*nScale,12.0*nScale,0];
        MoveL pTarget,vSpeed,z0,tTool\WObj:=wWobj;
        pTarget.trans:=[6*nScale,13.0*nScale,0];
        MoveL pTarget,vSpeed,z0,tTool\WObj:=wWobj;
        pTarget.trans:=[8*nScale,16.0*nScale,0];
        MoveL pTarget,vSpeed,fine,tTool\WObj:=wWobj;
        Reset do_pen;
        MoveL RelTool(pTarget,0,0,-2),vSpeed,z0,tTool\WObj:=wWobj;
        wWobj.oframe.trans.x:=wWobj.oframe.trans.x+8*nScale;
    ENDPROC

    ! Character: m
    PROC char_m(\num nScaleParam)
        VAR robtarget pTarget;
        VAR num nScale:=1;
        pTarget:=refTarget;
        IF Present(nScaleParam) THEN
            nScale:=nScaleParam;
        ENDIF
        pTarget.trans:=[0*nScale,16.0*nScale,0];
        MoveL pTarget,vSpeed,fine,tTool\WObj:=wWobj;
        Set do_pen;
        pTarget.trans:=[2*nScale,19.0*nScale,0];
        MoveL pTarget,vSpeed,z0,tTool\WObj:=wWobj;
        pTarget.trans:=[4*nScale,20.0*nScale,0];
        MoveL pTarget,vSpeed,z0,tTool\WObj:=wWobj;
        pTarget.trans:=[5*nScale,19.0*nScale,0];
        MoveL pTarget,vSpeed,z0,tTool\WObj:=wWobj;
        pTarget.trans:=[5*nScale,18.0*nScale,0];
        MoveL pTarget,vSpeed,z0,tTool\WObj:=wWobj;
        pTarget.trans:=[4*nScale,14.0*nScale,0];
        MoveL pTarget,vSpeed,z0,tTool\WObj:=wWobj;
        pTarget.trans:=[3*nScale,11.0*nScale,0];
        MoveL pTarget,vSpeed,fine,tTool\WObj:=wWobj;
        Reset do_pen;
        MoveL RelTool(pTarget,0,0,-2),vSpeed,z0,tTool\WObj:=wWobj;
        pTarget.trans:=[4*nScale,14.0*nScale,0];
        MoveL pTarget,vSpeed,fine,tTool\WObj:=wWobj;
        Set do_pen;
        pTarget.trans:=[5*nScale,16.0*nScale,0];
        MoveL pTarget,vSpeed,z0,tTool\WObj:=wWobj;
        pTarget.trans:=[7*nScale,19.0*nScale,0];
        MoveL pTarget,vSpeed,z0,tTool\WObj:=wWobj;
        pTarget.trans:=[9*nScale,20.0*nScale,0];
        MoveL pTarget,vSpeed,z0,tTool\WObj:=wWobj;
        pTarget.trans:=[11*nScale,20.0*nScale,0];
        MoveL pTarget,vSpeed,z0,tTool\WObj:=wWobj;
        pTarget.trans:=[12*nScale,19.0*nScale,0];
        MoveL pTarget,vSpeed,z0,tTool\WObj:=wWobj;
        pTarget.trans:=[12*nScale,18.0*nScale,0];
        MoveL pTarget,vSpeed,z0,tTool\WObj:=wWobj;
        pTarget.trans:=[11*nScale,14.0*nScale,0];
        MoveL pTarget,vSpeed,z0,tTool\WObj:=wWobj;
        pTarget.trans:=[10*nScale,11.0*nScale,0];
        MoveL pTarget,vSpeed,fine,tTool\WObj:=wWobj;
        Reset do_pen;
        MoveL RelTool(pTarget,0,0,-2),vSpeed,z0,tTool\WObj:=wWobj;
        pTarget.trans:=[11*nScale,14.0*nScale,0];
        MoveL pTarget,vSpeed,fine,tTool\WObj:=wWobj;
        Set do_pen;
        pTarget.trans:=[12*nScale,16.0*nScale,0];
        MoveL pTarget,vSpeed,z0,tTool\WObj:=wWobj;
        pTarget.trans:=[14*nScale,19.0*nScale,0];
        MoveL pTarget,vSpeed,z0,tTool\WObj:=wWobj;
        pTarget.trans:=[16*nScale,20.0*nScale,0];
        MoveL pTarget,vSpeed,z0,tTool\WObj:=wWobj;
        pTarget.trans:=[18*nScale,20.0*nScale,0];
        MoveL pTarget,vSpeed,z0,tTool\WObj:=wWobj;
        pTarget.trans:=[19*nScale,19.0*nScale,0];
        MoveL pTarget,vSpeed,z0,tTool\WObj:=wWobj;
        pTarget.trans:=[19*nScale,17.0*nScale,0];
        MoveL pTarget,vSpeed,z0,tTool\WObj:=wWobj;
        pTarget.trans:=[18*nScale,14.0*nScale,0];
        MoveL pTarget,vSpeed,z0,tTool\WObj:=wWobj;
        pTarget.trans:=[18*nScale,12.0*nScale,0];
        MoveL pTarget,vSpeed,z0,tTool\WObj:=wWobj;
        pTarget.trans:=[19*nScale,11.0*nScale,0];
        MoveL pTarget,vSpeed,z0,tTool\WObj:=wWobj;
        pTarget.trans:=[20*nScale,11.0*nScale,0];
        MoveL pTarget,vSpeed,z0,tTool\WObj:=wWobj;
        pTarget.trans:=[22*nScale,12.0*nScale,0];
        MoveL pTarget,vSpeed,z0,tTool\WObj:=wWobj;
        pTarget.trans:=[23*nScale,13.0*nScale,0];
        MoveL pTarget,vSpeed,z0,tTool\WObj:=wWobj;
        pTarget.trans:=[25*nScale,16.0*nScale,0];
        MoveL pTarget,vSpeed,fine,tTool\WObj:=wWobj;
        Reset do_pen;
        MoveL RelTool(pTarget,0,0,-2),vSpeed,z0,tTool\WObj:=wWobj;
        wWobj.oframe.trans.x:=wWobj.oframe.trans.x+25*nScale;
    ENDPROC

    ! Character: n
    PROC char_n(\num nScaleParam)
        VAR robtarget pTarget;
        VAR num nScale:=1;
        pTarget:=refTarget;
        IF Present(nScaleParam) THEN
            nScale:=nScaleParam;
        ENDIF
        pTarget.trans:=[0*nScale,16.0*nScale,0];
        MoveL pTarget,vSpeed,fine,tTool\WObj:=wWobj;
        Set do_pen;
        pTarget.trans:=[2*nScale,19.0*nScale,0];
        MoveL pTarget,vSpeed,z0,tTool\WObj:=wWobj;
        pTarget.trans:=[4*nScale,20.0*nScale,0];
        MoveL pTarget,vSpeed,z0,tTool\WObj:=wWobj;
        pTarget.trans:=[5*nScale,19.0*nScale,0];
        MoveL pTarget,vSpeed,z0,tTool\WObj:=wWobj;
        pTarget.trans:=[5*nScale,18.0*nScale,0];
        MoveL pTarget,vSpeed,z0,tTool\WObj:=wWobj;
        pTarget.trans:=[4*nScale,14.0*nScale,0];
        MoveL pTarget,vSpeed,z0,tTool\WObj:=wWobj;
        pTarget.trans:=[3*nScale,11.0*nScale,0];
        MoveL pTarget,vSpeed,fine,tTool\WObj:=wWobj;
        Reset do_pen;
        MoveL RelTool(pTarget,0,0,-2),vSpeed,z0,tTool\WObj:=wWobj;
        pTarget.trans:=[4*nScale,14.0*nScale,0];
        MoveL pTarget,vSpeed,fine,tTool\WObj:=wWobj;
        Set do_pen;
        pTarget.trans:=[5*nScale,16.0*nScale,0];
        MoveL pTarget,vSpeed,z0,tTool\WObj:=wWobj;
        pTarget.trans:=[7*nScale,19.0*nScale,0];
        MoveL pTarget,vSpeed,z0,tTool\WObj:=wWobj;
        pTarget.trans:=[9*nScale,20.0*nScale,0];
        MoveL pTarget,vSpeed,z0,tTool\WObj:=wWobj;
        pTarget.trans:=[11*nScale,20.0*nScale,0];
        MoveL pTarget,vSpeed,z0,tTool\WObj:=wWobj;
        pTarget.trans:=[12*nScale,19.0*nScale,0];
        MoveL pTarget,vSpeed,z0,tTool\WObj:=wWobj;
        pTarget.trans:=[12*nScale,17.0*nScale,0];
        MoveL pTarget,vSpeed,z0,tTool\WObj:=wWobj;
        pTarget.trans:=[11*nScale,14.0*nScale,0];
        MoveL pTarget,vSpeed,z0,tTool\WObj:=wWobj;
        pTarget.trans:=[11*nScale,12.0*nScale,0];
        MoveL pTarget,vSpeed,z0,tTool\WObj:=wWobj;
        pTarget.trans:=[12*nScale,11.0*nScale,0];
        MoveL pTarget,vSpeed,z0,tTool\WObj:=wWobj;
        pTarget.trans:=[13*nScale,11.0*nScale,0];
        MoveL pTarget,vSpeed,z0,tTool\WObj:=wWobj;
        pTarget.trans:=[15*nScale,12.0*nScale,0];
        MoveL pTarget,vSpeed,z0,tTool\WObj:=wWobj;
        pTarget.trans:=[16*nScale,13.0*nScale,0];
        MoveL pTarget,vSpeed,z0,tTool\WObj:=wWobj;
        pTarget.trans:=[18*nScale,16.0*nScale,0];
        MoveL pTarget,vSpeed,fine,tTool\WObj:=wWobj;
        Reset do_pen;
        MoveL RelTool(pTarget,0,0,-2),vSpeed,z0,tTool\WObj:=wWobj;
        wWobj.oframe.trans.x:=wWobj.oframe.trans.x+18*nScale;
    ENDPROC

    ! Character: o
    PROC char_o(\num nScaleParam)
        VAR robtarget pTarget;
        VAR num nScale:=1;
        pTarget:=refTarget;
        IF Present(nScaleParam) THEN
            nScale:=nScaleParam;
        ENDIF
        pTarget.trans:=[6*nScale,20.0*nScale,0];
        MoveL pTarget,vSpeed,fine,tTool\WObj:=wWobj;
        Set do_pen;
        pTarget.trans:=[4*nScale,20.0*nScale,0];
        MoveL pTarget,vSpeed,z0,tTool\WObj:=wWobj;
        pTarget.trans:=[2*nScale,19.0*nScale,0];
        MoveL pTarget,vSpeed,z0,tTool\WObj:=wWobj;
        pTarget.trans:=[1*nScale,18.0*nScale,0];
        MoveL pTarget,vSpeed,z0,tTool\WObj:=wWobj;
        pTarget.trans:=[0*nScale,16.0*nScale,0];
        MoveL pTarget,vSpeed,z0,tTool\WObj:=wWobj;
        pTarget.trans:=[0*nScale,14.0*nScale,0];
        MoveL pTarget,vSpeed,z0,tTool\WObj:=wWobj;
        pTarget.trans:=[1*nScale,12.0*nScale,0];
        MoveL pTarget,vSpeed,z0,tTool\WObj:=wWobj;
        pTarget.trans:=[3*nScale,11.0*nScale,0];
        MoveL pTarget,vSpeed,z0,tTool\WObj:=wWobj;
        pTarget.trans:=[5*nScale,11.0*nScale,0];
        MoveL pTarget,vSpeed,z0,tTool\WObj:=wWobj;
        pTarget.trans:=[7*nScale,12.0*nScale,0];
        MoveL pTarget,vSpeed,z0,tTool\WObj:=wWobj;
        pTarget.trans:=[8*nScale,13.0*nScale,0];
        MoveL pTarget,vSpeed,z0,tTool\WObj:=wWobj;
        pTarget.trans:=[9*nScale,15.0*nScale,0];
        MoveL pTarget,vSpeed,z0,tTool\WObj:=wWobj;
        pTarget.trans:=[9*nScale,17.0*nScale,0];
        MoveL pTarget,vSpeed,z0,tTool\WObj:=wWobj;
        pTarget.trans:=[8*nScale,19.0*nScale,0];
        MoveL pTarget,vSpeed,z0,tTool\WObj:=wWobj;
        pTarget.trans:=[6*nScale,20.0*nScale,0];
        MoveL pTarget,vSpeed,z0,tTool\WObj:=wWobj;
        pTarget.trans:=[5*nScale,19.0*nScale,0];
        MoveL pTarget,vSpeed,z0,tTool\WObj:=wWobj;
        pTarget.trans:=[5*nScale,17.0*nScale,0];
        MoveL pTarget,vSpeed,z0,tTool\WObj:=wWobj;
        pTarget.trans:=[6*nScale,15.0*nScale,0];
        MoveL pTarget,vSpeed,z0,tTool\WObj:=wWobj;
        pTarget.trans:=[8*nScale,14.0*nScale,0];
        MoveL pTarget,vSpeed,z0,tTool\WObj:=wWobj;
        pTarget.trans:=[11*nScale,14.0*nScale,0];
        MoveL pTarget,vSpeed,z0,tTool\WObj:=wWobj;
        pTarget.trans:=[13*nScale,15.0*nScale,0];
        MoveL pTarget,vSpeed,z0,tTool\WObj:=wWobj;
        pTarget.trans:=[14*nScale,16.0*nScale,0];
        MoveL pTarget,vSpeed,fine,tTool\WObj:=wWobj;
        Reset do_pen;
        MoveL RelTool(pTarget,0,0,-2),vSpeed,z0,tTool\WObj:=wWobj;
        wWobj.oframe.trans.x:=wWobj.oframe.trans.x+14*nScale;
    ENDPROC

    ! Character: p
    PROC char_p(\num nScaleParam)
        VAR robtarget pTarget;
        VAR num nScale:=1;
        pTarget:=refTarget;
        IF Present(nScaleParam) THEN
            nScale:=nScaleParam;
        ENDIF
        pTarget.trans:=[0*nScale,16.0*nScale,0];
        MoveL pTarget,vSpeed,fine,tTool\WObj:=wWobj;
        Set do_pen;
        pTarget.trans:=[2*nScale,19.0*nScale,0];
        MoveL pTarget,vSpeed,z0,tTool\WObj:=wWobj;
        pTarget.trans:=[3*nScale,21.0*nScale,0];
        MoveL pTarget,vSpeed,z0,tTool\WObj:=wWobj;
        pTarget.trans:=[2*nScale,17.0*nScale,0];
        MoveL pTarget,vSpeed,z0,tTool\WObj:=wWobj;
        pTarget.trans:=[-4*nScale,-1.0*nScale,0];
        MoveL pTarget,vSpeed,fine,tTool\WObj:=wWobj;
        Reset do_pen;
        MoveL RelTool(pTarget,0,0,-2),vSpeed,z0,tTool\WObj:=wWobj;
        pTarget.trans:=[2*nScale,17.0*nScale,0];
        MoveL pTarget,vSpeed,fine,tTool\WObj:=wWobj;
        Set do_pen;
        pTarget.trans:=[3*nScale,19.0*nScale,0];
        MoveL pTarget,vSpeed,z0,tTool\WObj:=wWobj;
        pTarget.trans:=[5*nScale,20.0*nScale,0];
        MoveL pTarget,vSpeed,z0,tTool\WObj:=wWobj;
        pTarget.trans:=[7*nScale,20.0*nScale,0];
        MoveL pTarget,vSpeed,z0,tTool\WObj:=wWobj;
        pTarget.trans:=[9*nScale,19.0*nScale,0];
        MoveL pTarget,vSpeed,z0,tTool\WObj:=wWobj;
        pTarget.trans:=[10*nScale,17.0*nScale,0];
        MoveL pTarget,vSpeed,z0,tTool\WObj:=wWobj;
        pTarget.trans:=[10*nScale,15.0*nScale,0];
        MoveL pTarget,vSpeed,z0,tTool\WObj:=wWobj;
        pTarget.trans:=[9*nScale,13.0*nScale,0];
        MoveL pTarget,vSpeed,z0,tTool\WObj:=wWobj;
        pTarget.trans:=[8*nScale,12.0*nScale,0];
        MoveL pTarget,vSpeed,z0,tTool\WObj:=wWobj;
        pTarget.trans:=[6*nScale,11.0*nScale,0];
        MoveL pTarget,vSpeed,fine,tTool\WObj:=wWobj;
        Reset do_pen;
        MoveL RelTool(pTarget,0,0,-2),vSpeed,z0,tTool\WObj:=wWobj;
        pTarget.trans:=[2*nScale,12.0*nScale,0];
        MoveL pTarget,vSpeed,fine,tTool\WObj:=wWobj;
        Set do_pen;
        pTarget.trans:=[4*nScale,11.0*nScale,0];
        MoveL pTarget,vSpeed,z0,tTool\WObj:=wWobj;
        pTarget.trans:=[7*nScale,11.0*nScale,0];
        MoveL pTarget,vSpeed,z0,tTool\WObj:=wWobj;
        pTarget.trans:=[10*nScale,12.0*nScale,0];
        MoveL pTarget,vSpeed,z0,tTool\WObj:=wWobj;
        pTarget.trans:=[12*nScale,13.0*nScale,0];
        MoveL pTarget,vSpeed,z0,tTool\WObj:=wWobj;
        pTarget.trans:=[15*nScale,16.0*nScale,0];
        MoveL pTarget,vSpeed,fine,tTool\WObj:=wWobj;
        Reset do_pen;
        MoveL RelTool(pTarget,0,0,-2),vSpeed,z0,tTool\WObj:=wWobj;
        wWobj.oframe.trans.x:=wWobj.oframe.trans.x+15*nScale;
    ENDPROC

    ! Character: q
    PROC char_q(\num nScaleParam)
        VAR robtarget pTarget;
        VAR num nScale:=1;
        pTarget:=refTarget;
        IF Present(nScaleParam) THEN
            nScale:=nScaleParam;
        ENDIF
        pTarget.trans:=[9*nScale,17.0*nScale,0];
        MoveL pTarget,vSpeed,fine,tTool\WObj:=wWobj;
        Set do_pen;
        pTarget.trans:=[8*nScale,19.0*nScale,0];
        MoveL pTarget,vSpeed,z0,tTool\WObj:=wWobj;
        pTarget.trans:=[6*nScale,20.0*nScale,0];
        MoveL pTarget,vSpeed,z0,tTool\WObj:=wWobj;
        pTarget.trans:=[4*nScale,20.0*nScale,0];
        MoveL pTarget,vSpeed,z0,tTool\WObj:=wWobj;
        pTarget.trans:=[2*nScale,19.0*nScale,0];
        MoveL pTarget,vSpeed,z0,tTool\WObj:=wWobj;
        pTarget.trans:=[1*nScale,18.0*nScale,0];
        MoveL pTarget,vSpeed,z0,tTool\WObj:=wWobj;
        pTarget.trans:=[0*nScale,16.0*nScale,0];
        MoveL pTarget,vSpeed,z0,tTool\WObj:=wWobj;
        pTarget.trans:=[0*nScale,14.0*nScale,0];
        MoveL pTarget,vSpeed,z0,tTool\WObj:=wWobj;
        pTarget.trans:=[1*nScale,12.0*nScale,0];
        MoveL pTarget,vSpeed,z0,tTool\WObj:=wWobj;
        pTarget.trans:=[3*nScale,11.0*nScale,0];
        MoveL pTarget,vSpeed,z0,tTool\WObj:=wWobj;
        pTarget.trans:=[5*nScale,11.0*nScale,0];
        MoveL pTarget,vSpeed,z0,tTool\WObj:=wWobj;
        pTarget.trans:=[7*nScale,12.0*nScale,0];
        MoveL pTarget,vSpeed,fine,tTool\WObj:=wWobj;
        Reset do_pen;
        MoveL RelTool(pTarget,0,0,-2),vSpeed,z0,tTool\WObj:=wWobj;
        pTarget.trans:=[10*nScale,20.0*nScale,0];
        MoveL pTarget,vSpeed,fine,tTool\WObj:=wWobj;
        Set do_pen;
        pTarget.trans:=[9*nScale,17.0*nScale,0];
        MoveL pTarget,vSpeed,z0,tTool\WObj:=wWobj;
        pTarget.trans:=[7*nScale,12.0*nScale,0];
        MoveL pTarget,vSpeed,z0,tTool\WObj:=wWobj;
        pTarget.trans:=[4*nScale,5.0*nScale,0];
        MoveL pTarget,vSpeed,z0,tTool\WObj:=wWobj;
        pTarget.trans:=[3*nScale,2.0*nScale,0];
        MoveL pTarget,vSpeed,z0,tTool\WObj:=wWobj;
        pTarget.trans:=[3*nScale,0.0*nScale,0];
        MoveL pTarget,vSpeed,z0,tTool\WObj:=wWobj;
        pTarget.trans:=[4*nScale,-1.0*nScale,0];
        MoveL pTarget,vSpeed,z0,tTool\WObj:=wWobj;
        pTarget.trans:=[6*nScale,0.0*nScale,0];
        MoveL pTarget,vSpeed,z0,tTool\WObj:=wWobj;
        pTarget.trans:=[7*nScale,3.0*nScale,0];
        MoveL pTarget,vSpeed,z0,tTool\WObj:=wWobj;
        pTarget.trans:=[7*nScale,10.0*nScale,0];
        MoveL pTarget,vSpeed,z0,tTool\WObj:=wWobj;
        pTarget.trans:=[9*nScale,11.0*nScale,0];
        MoveL pTarget,vSpeed,z0,tTool\WObj:=wWobj;
        pTarget.trans:=[12*nScale,13.0*nScale,0];
        MoveL pTarget,vSpeed,z0,tTool\WObj:=wWobj;
        pTarget.trans:=[15*nScale,16.0*nScale,0];
        MoveL pTarget,vSpeed,fine,tTool\WObj:=wWobj;
        Reset do_pen;
        MoveL RelTool(pTarget,0,0,-2),vSpeed,z0,tTool\WObj:=wWobj;
        wWobj.oframe.trans.x:=wWobj.oframe.trans.x+15*nScale;
    ENDPROC

    ! Character: r
    PROC char_r(\num nScaleParam)
        VAR robtarget pTarget;
        VAR num nScale:=1;
        pTarget:=refTarget;
        IF Present(nScaleParam) THEN
            nScale:=nScaleParam;
        ENDIF
        pTarget.trans:=[0*nScale,16.0*nScale,0];
        MoveL pTarget,vSpeed,fine,tTool\WObj:=wWobj;
        Set do_pen;
        pTarget.trans:=[2*nScale,19.0*nScale,0];
        MoveL pTarget,vSpeed,z0,tTool\WObj:=wWobj;
        pTarget.trans:=[3*nScale,21.0*nScale,0];
        MoveL pTarget,vSpeed,z0,tTool\WObj:=wWobj;
        pTarget.trans:=[3*nScale,19.0*nScale,0];
        MoveL pTarget,vSpeed,z0,tTool\WObj:=wWobj;
        pTarget.trans:=[6*nScale,19.0*nScale,0];
        MoveL pTarget,vSpeed,z0,tTool\WObj:=wWobj;
        pTarget.trans:=[7*nScale,18.0*nScale,0];
        MoveL pTarget,vSpeed,z0,tTool\WObj:=wWobj;
        pTarget.trans:=[7*nScale,16.0*nScale,0];
        MoveL pTarget,vSpeed,z0,tTool\WObj:=wWobj;
        pTarget.trans:=[6*nScale,13.0*nScale,0];
        MoveL pTarget,vSpeed,z0,tTool\WObj:=wWobj;
        pTarget.trans:=[6*nScale,12.0*nScale,0];
        MoveL pTarget,vSpeed,z0,tTool\WObj:=wWobj;
        pTarget.trans:=[7*nScale,11.0*nScale,0];
        MoveL pTarget,vSpeed,z0,tTool\WObj:=wWobj;
        pTarget.trans:=[8*nScale,11.0*nScale,0];
        MoveL pTarget,vSpeed,z0,tTool\WObj:=wWobj;
        pTarget.trans:=[10*nScale,12.0*nScale,0];
        MoveL pTarget,vSpeed,z0,tTool\WObj:=wWobj;
        pTarget.trans:=[11*nScale,13.0*nScale,0];
        MoveL pTarget,vSpeed,z0,tTool\WObj:=wWobj;
        pTarget.trans:=[13*nScale,16.0*nScale,0];
        MoveL pTarget,vSpeed,fine,tTool\WObj:=wWobj;
        Reset do_pen;
        MoveL RelTool(pTarget,0,0,-2),vSpeed,z0,tTool\WObj:=wWobj;
        wWobj.oframe.trans.x:=wWobj.oframe.trans.x+13*nScale;
    ENDPROC

    ! Character: s
    PROC char_s(\num nScaleParam)
        VAR robtarget pTarget;
        VAR num nScale:=1;
        pTarget:=refTarget;
        IF Present(nScaleParam) THEN
            nScale:=nScaleParam;
        ENDIF
        pTarget.trans:=[0*nScale,16.0*nScale,0];
        MoveL pTarget,vSpeed,fine,tTool\WObj:=wWobj;
        Set do_pen;
        pTarget.trans:=[2*nScale,19.0*nScale,0];
        MoveL pTarget,vSpeed,z0,tTool\WObj:=wWobj;
        pTarget.trans:=[3*nScale,21.0*nScale,0];
        MoveL pTarget,vSpeed,z0,tTool\WObj:=wWobj;
        pTarget.trans:=[3*nScale,19.0*nScale,0];
        MoveL pTarget,vSpeed,z0,tTool\WObj:=wWobj;
        pTarget.trans:=[5*nScale,16.0*nScale,0];
        MoveL pTarget,vSpeed,z0,tTool\WObj:=wWobj;
        pTarget.trans:=[6*nScale,14.0*nScale,0];
        MoveL pTarget,vSpeed,z0,tTool\WObj:=wWobj;
        pTarget.trans:=[6*nScale,12.0*nScale,0];
        MoveL pTarget,vSpeed,z0,tTool\WObj:=wWobj;
        pTarget.trans:=[4*nScale,11.0*nScale,0];
        MoveL pTarget,vSpeed,fine,tTool\WObj:=wWobj;
        Reset do_pen;
        MoveL RelTool(pTarget,0,0,-2),vSpeed,z0,tTool\WObj:=wWobj;
        pTarget.trans:=[0*nScale,12.0*nScale,0];
        MoveL pTarget,vSpeed,fine,tTool\WObj:=wWobj;
        Set do_pen;
        pTarget.trans:=[2*nScale,11.0*nScale,0];
        MoveL pTarget,vSpeed,z0,tTool\WObj:=wWobj;
        pTarget.trans:=[6*nScale,11.0*nScale,0];
        MoveL pTarget,vSpeed,z0,tTool\WObj:=wWobj;
        pTarget.trans:=[8*nScale,12.0*nScale,0];
        MoveL pTarget,vSpeed,z0,tTool\WObj:=wWobj;
        pTarget.trans:=[9*nScale,13.0*nScale,0];
        MoveL pTarget,vSpeed,z0,tTool\WObj:=wWobj;
        pTarget.trans:=[11*nScale,16.0*nScale,0];
        MoveL pTarget,vSpeed,fine,tTool\WObj:=wWobj;
        Reset do_pen;
        MoveL RelTool(pTarget,0,0,-2),vSpeed,z0,tTool\WObj:=wWobj;
        wWobj.oframe.trans.x:=wWobj.oframe.trans.x+11*nScale;
    ENDPROC

    ! Character: t
    PROC char_t(\num nScaleParam)
        VAR robtarget pTarget;
        VAR num nScale:=1;
        pTarget:=refTarget;
        IF Present(nScaleParam) THEN
            nScale:=nScaleParam;
        ENDIF
        pTarget.trans:=[0*nScale,16.0*nScale,0];
        MoveL pTarget,vSpeed,fine,tTool\WObj:=wWobj;
        Set do_pen;
        pTarget.trans:=[2*nScale,19.0*nScale,0];
        MoveL pTarget,vSpeed,z0,tTool\WObj:=wWobj;
        pTarget.trans:=[4*nScale,23.0*nScale,0];
        MoveL pTarget,vSpeed,fine,tTool\WObj:=wWobj;
        Reset do_pen;
        MoveL RelTool(pTarget,0,0,-2),vSpeed,z0,tTool\WObj:=wWobj;
        pTarget.trans:=[7*nScale,32.0*nScale,0];
        MoveL pTarget,vSpeed,fine,tTool\WObj:=wWobj;
        Set do_pen;
        pTarget.trans:=[1*nScale,14.0*nScale,0];
        MoveL pTarget,vSpeed,z0,tTool\WObj:=wWobj;
        pTarget.trans:=[1*nScale,12.0*nScale,0];
        MoveL pTarget,vSpeed,z0,tTool\WObj:=wWobj;
        pTarget.trans:=[2*nScale,11.0*nScale,0];
        MoveL pTarget,vSpeed,z0,tTool\WObj:=wWobj;
        pTarget.trans:=[4*nScale,11.0*nScale,0];
        MoveL pTarget,vSpeed,z0,tTool\WObj:=wWobj;
        pTarget.trans:=[6*nScale,12.0*nScale,0];
        MoveL pTarget,vSpeed,z0,tTool\WObj:=wWobj;
        pTarget.trans:=[7*nScale,13.0*nScale,0];
        MoveL pTarget,vSpeed,z0,tTool\WObj:=wWobj;
        pTarget.trans:=[9*nScale,16.0*nScale,0];
        MoveL pTarget,vSpeed,fine,tTool\WObj:=wWobj;
        Reset do_pen;
        MoveL RelTool(pTarget,0,0,-2),vSpeed,z0,tTool\WObj:=wWobj;
        pTarget.trans:=[1*nScale,24.0*nScale,0];
        MoveL pTarget,vSpeed,fine,tTool\WObj:=wWobj;
        Set do_pen;
        pTarget.trans:=[8*nScale,24.0*nScale,0];
        MoveL pTarget,vSpeed,fine,tTool\WObj:=wWobj;
        Reset do_pen;
        MoveL RelTool(pTarget,0,0,-2),vSpeed,z0,tTool\WObj:=wWobj;
        wWobj.oframe.trans.x:=wWobj.oframe.trans.x+9*nScale;
    ENDPROC

    ! Character: u
    PROC char_u(\num nScaleParam)
        VAR robtarget pTarget;
        VAR num nScale:=1;
        pTarget:=refTarget;
        IF Present(nScaleParam) THEN
            nScale:=nScaleParam;
        ENDIF
        pTarget.trans:=[0*nScale,16.0*nScale,0];
        MoveL pTarget,vSpeed,fine,tTool\WObj:=wWobj;
        Set do_pen;
        pTarget.trans:=[2*nScale,20.0*nScale,0];
        MoveL pTarget,vSpeed,z0,tTool\WObj:=wWobj;
        pTarget.trans:=[0*nScale,14.0*nScale,0];
        MoveL pTarget,vSpeed,z0,tTool\WObj:=wWobj;
        pTarget.trans:=[0*nScale,12.0*nScale,0];
        MoveL pTarget,vSpeed,z0,tTool\WObj:=wWobj;
        pTarget.trans:=[1*nScale,11.0*nScale,0];
        MoveL pTarget,vSpeed,z0,tTool\WObj:=wWobj;
        pTarget.trans:=[3*nScale,11.0*nScale,0];
        MoveL pTarget,vSpeed,z0,tTool\WObj:=wWobj;
        pTarget.trans:=[5*nScale,12.0*nScale,0];
        MoveL pTarget,vSpeed,z0,tTool\WObj:=wWobj;
        pTarget.trans:=[7*nScale,14.0*nScale,0];
        MoveL pTarget,vSpeed,z0,tTool\WObj:=wWobj;
        pTarget.trans:=[9*nScale,17.0*nScale,0];
        MoveL pTarget,vSpeed,fine,tTool\WObj:=wWobj;
        Reset do_pen;
        MoveL RelTool(pTarget,0,0,-2),vSpeed,z0,tTool\WObj:=wWobj;
        pTarget.trans:=[10*nScale,20.0*nScale,0];
        MoveL pTarget,vSpeed,fine,tTool\WObj:=wWobj;
        Set do_pen;
        pTarget.trans:=[8*nScale,14.0*nScale,0];
        MoveL pTarget,vSpeed,z0,tTool\WObj:=wWobj;
        pTarget.trans:=[8*nScale,12.0*nScale,0];
        MoveL pTarget,vSpeed,z0,tTool\WObj:=wWobj;
        pTarget.trans:=[9*nScale,11.0*nScale,0];
        MoveL pTarget,vSpeed,z0,tTool\WObj:=wWobj;
        pTarget.trans:=[10*nScale,11.0*nScale,0];
        MoveL pTarget,vSpeed,z0,tTool\WObj:=wWobj;
        pTarget.trans:=[12*nScale,12.0*nScale,0];
        MoveL pTarget,vSpeed,z0,tTool\WObj:=wWobj;
        pTarget.trans:=[13*nScale,13.0*nScale,0];
        MoveL pTarget,vSpeed,z0,tTool\WObj:=wWobj;
        pTarget.trans:=[15*nScale,16.0*nScale,0];
        MoveL pTarget,vSpeed,fine,tTool\WObj:=wWobj;
        Reset do_pen;
        MoveL RelTool(pTarget,0,0,-2),vSpeed,z0,tTool\WObj:=wWobj;
        wWobj.oframe.trans.x:=wWobj.oframe.trans.x+15*nScale;
    ENDPROC

    ! Character: v
    PROC char_v(\num nScaleParam)
        VAR robtarget pTarget;
        VAR num nScale:=1;
        pTarget:=refTarget;
        IF Present(nScaleParam) THEN
            nScale:=nScaleParam;
        ENDIF
        pTarget.trans:=[0*nScale,16.0*nScale,0];
        MoveL pTarget,vSpeed,fine,tTool\WObj:=wWobj;
        Set do_pen;
        pTarget.trans:=[2*nScale,20.0*nScale,0];
        MoveL pTarget,vSpeed,z0,tTool\WObj:=wWobj;
        pTarget.trans:=[1*nScale,15.0*nScale,0];
        MoveL pTarget,vSpeed,z0,tTool\WObj:=wWobj;
        pTarget.trans:=[1*nScale,12.0*nScale,0];
        MoveL pTarget,vSpeed,z0,tTool\WObj:=wWobj;
        pTarget.trans:=[2*nScale,11.0*nScale,0];
        MoveL pTarget,vSpeed,z0,tTool\WObj:=wWobj;
        pTarget.trans:=[3*nScale,11.0*nScale,0];
        MoveL pTarget,vSpeed,z0,tTool\WObj:=wWobj;
        pTarget.trans:=[6*nScale,12.0*nScale,0];
        MoveL pTarget,vSpeed,z0,tTool\WObj:=wWobj;
        pTarget.trans:=[8*nScale,14.0*nScale,0];
        MoveL pTarget,vSpeed,z0,tTool\WObj:=wWobj;
        pTarget.trans:=[9*nScale,17.0*nScale,0];
        MoveL pTarget,vSpeed,z0,tTool\WObj:=wWobj;
        pTarget.trans:=[9*nScale,20.0*nScale,0];
        MoveL pTarget,vSpeed,fine,tTool\WObj:=wWobj;
        Reset do_pen;
        MoveL RelTool(pTarget,0,0,-2),vSpeed,z0,tTool\WObj:=wWobj;
        pTarget.trans:=[9*nScale,20.0*nScale,0];
        MoveL pTarget,vSpeed,fine,tTool\WObj:=wWobj;
        Set do_pen;
        pTarget.trans:=[10*nScale,16.0*nScale,0];
        MoveL pTarget,vSpeed,z0,tTool\WObj:=wWobj;
        pTarget.trans:=[11*nScale,15.0*nScale,0];
        MoveL pTarget,vSpeed,z0,tTool\WObj:=wWobj;
        pTarget.trans:=[13*nScale,15.0*nScale,0];
        MoveL pTarget,vSpeed,z0,tTool\WObj:=wWobj;
        pTarget.trans:=[15*nScale,16.0*nScale,0];
        MoveL pTarget,vSpeed,fine,tTool\WObj:=wWobj;
        Reset do_pen;
        MoveL RelTool(pTarget,0,0,-2),vSpeed,z0,tTool\WObj:=wWobj;
        wWobj.oframe.trans.x:=wWobj.oframe.trans.x+15*nScale;
    ENDPROC

    ! Character: w
    PROC char_w(\num nScaleParam)
        VAR robtarget pTarget;
        VAR num nScale:=1;
        pTarget:=refTarget;
        IF Present(nScaleParam) THEN
            nScale:=nScaleParam;
        ENDIF
        pTarget.trans:=[3*nScale,20.0*nScale,0];
        MoveL pTarget,vSpeed,fine,tTool\WObj:=wWobj;
        Set do_pen;
        pTarget.trans:=[1*nScale,18.0*nScale,0];
        MoveL pTarget,vSpeed,z0,tTool\WObj:=wWobj;
        pTarget.trans:=[0*nScale,15.0*nScale,0];
        MoveL pTarget,vSpeed,z0,tTool\WObj:=wWobj;
        pTarget.trans:=[0*nScale,13.0*nScale,0];
        MoveL pTarget,vSpeed,z0,tTool\WObj:=wWobj;
        pTarget.trans:=[1*nScale,11.0*nScale,0];
        MoveL pTarget,vSpeed,z0,tTool\WObj:=wWobj;
        pTarget.trans:=[3*nScale,11.0*nScale,0];
        MoveL pTarget,vSpeed,z0,tTool\WObj:=wWobj;
        pTarget.trans:=[5*nScale,12.0*nScale,0];
        MoveL pTarget,vSpeed,z0,tTool\WObj:=wWobj;
        pTarget.trans:=[7*nScale,14.0*nScale,0];
        MoveL pTarget,vSpeed,fine,tTool\WObj:=wWobj;
        Reset do_pen;
        MoveL RelTool(pTarget,0,0,-2),vSpeed,z0,tTool\WObj:=wWobj;
        pTarget.trans:=[9*nScale,20.0*nScale,0];
        MoveL pTarget,vSpeed,fine,tTool\WObj:=wWobj;
        Set do_pen;
        pTarget.trans:=[7*nScale,14.0*nScale,0];
        MoveL pTarget,vSpeed,z0,tTool\WObj:=wWobj;
        pTarget.trans:=[7*nScale,12.0*nScale,0];
        MoveL pTarget,vSpeed,z0,tTool\WObj:=wWobj;
        pTarget.trans:=[8*nScale,11.0*nScale,0];
        MoveL pTarget,vSpeed,z0,tTool\WObj:=wWobj;
        pTarget.trans:=[10*nScale,11.0*nScale,0];
        MoveL pTarget,vSpeed,z0,tTool\WObj:=wWobj;
        pTarget.trans:=[12*nScale,12.0*nScale,0];
        MoveL pTarget,vSpeed,z0,tTool\WObj:=wWobj;
        pTarget.trans:=[14*nScale,14.0*nScale,0];
        MoveL pTarget,vSpeed,z0,tTool\WObj:=wWobj;
        pTarget.trans:=[15*nScale,17.0*nScale,0];
        MoveL pTarget,vSpeed,z0,tTool\WObj:=wWobj;
        pTarget.trans:=[15*nScale,20.0*nScale,0];
        MoveL pTarget,vSpeed,fine,tTool\WObj:=wWobj;
        Reset do_pen;
        MoveL RelTool(pTarget,0,0,-2),vSpeed,z0,tTool\WObj:=wWobj;
        pTarget.trans:=[15*nScale,20.0*nScale,0];
        MoveL pTarget,vSpeed,fine,tTool\WObj:=wWobj;
        Set do_pen;
        pTarget.trans:=[16*nScale,16.0*nScale,0];
        MoveL pTarget,vSpeed,z0,tTool\WObj:=wWobj;
        pTarget.trans:=[17*nScale,15.0*nScale,0];
        MoveL pTarget,vSpeed,z0,tTool\WObj:=wWobj;
        pTarget.trans:=[19*nScale,15.0*nScale,0];
        MoveL pTarget,vSpeed,z0,tTool\WObj:=wWobj;
        pTarget.trans:=[21*nScale,16.0*nScale,0];
        MoveL pTarget,vSpeed,fine,tTool\WObj:=wWobj;
        Reset do_pen;
        MoveL RelTool(pTarget,0,0,-2),vSpeed,z0,tTool\WObj:=wWobj;
        wWobj.oframe.trans.x:=wWobj.oframe.trans.x+21*nScale;
    ENDPROC

    ! Character: x
    PROC char_x(\num nScaleParam)
        VAR robtarget pTarget;
        VAR num nScale:=1;
        pTarget:=refTarget;
        IF Present(nScaleParam) THEN
            nScale:=nScaleParam;
        ENDIF
        pTarget.trans:=[0*nScale,16.0*nScale,0];
        MoveL pTarget,vSpeed,fine,tTool\WObj:=wWobj;
        Set do_pen;
        pTarget.trans:=[2*nScale,19.0*nScale,0];
        MoveL pTarget,vSpeed,z0,tTool\WObj:=wWobj;
        pTarget.trans:=[4*nScale,20.0*nScale,0];
        MoveL pTarget,vSpeed,z0,tTool\WObj:=wWobj;
        pTarget.trans:=[6*nScale,20.0*nScale,0];
        MoveL pTarget,vSpeed,z0,tTool\WObj:=wWobj;
        pTarget.trans:=[7*nScale,19.0*nScale,0];
        MoveL pTarget,vSpeed,z0,tTool\WObj:=wWobj;
        pTarget.trans:=[7*nScale,12.0*nScale,0];
        MoveL pTarget,vSpeed,z0,tTool\WObj:=wWobj;
        pTarget.trans:=[8*nScale,11.0*nScale,0];
        MoveL pTarget,vSpeed,z0,tTool\WObj:=wWobj;
        pTarget.trans:=[11*nScale,11.0*nScale,0];
        MoveL pTarget,vSpeed,z0,tTool\WObj:=wWobj;
        pTarget.trans:=[14*nScale,13.0*nScale,0];
        MoveL pTarget,vSpeed,z0,tTool\WObj:=wWobj;
        pTarget.trans:=[16*nScale,16.0*nScale,0];
        MoveL pTarget,vSpeed,fine,tTool\WObj:=wWobj;
        Reset do_pen;
        MoveL RelTool(pTarget,0,0,-2),vSpeed,z0,tTool\WObj:=wWobj;
        pTarget.trans:=[13*nScale,19.0*nScale,0];
        MoveL pTarget,vSpeed,fine,tTool\WObj:=wWobj;
        Set do_pen;
        pTarget.trans:=[12*nScale,20.0*nScale,0];
        MoveL pTarget,vSpeed,z0,tTool\WObj:=wWobj;
        pTarget.trans:=[10*nScale,20.0*nScale,0];
        MoveL pTarget,vSpeed,z0,tTool\WObj:=wWobj;
        pTarget.trans:=[9*nScale,19.0*nScale,0];
        MoveL pTarget,vSpeed,z0,tTool\WObj:=wWobj;
        pTarget.trans:=[5*nScale,12.0*nScale,0];
        MoveL pTarget,vSpeed,z0,tTool\WObj:=wWobj;
        pTarget.trans:=[4*nScale,11.0*nScale,0];
        MoveL pTarget,vSpeed,z0,tTool\WObj:=wWobj;
        pTarget.trans:=[2*nScale,11.0*nScale,0];
        MoveL pTarget,vSpeed,z0,tTool\WObj:=wWobj;
        pTarget.trans:=[1*nScale,12.0*nScale,0];
        MoveL pTarget,vSpeed,fine,tTool\WObj:=wWobj;
        Reset do_pen;
        MoveL RelTool(pTarget,0,0,-2),vSpeed,z0,tTool\WObj:=wWobj;
        wWobj.oframe.trans.x:=wWobj.oframe.trans.x+16*nScale;
    ENDPROC

    ! Character: y
    PROC char_y(\num nScaleParam)
        VAR robtarget pTarget;
        VAR num nScale:=1;
        pTarget:=refTarget;
        IF Present(nScaleParam) THEN
            nScale:=nScaleParam;
        ENDIF
        pTarget.trans:=[0*nScale,16.0*nScale,0];
        MoveL pTarget,vSpeed,fine,tTool\WObj:=wWobj;
        Set do_pen;
        pTarget.trans:=[2*nScale,20.0*nScale,0];
        MoveL pTarget,vSpeed,z0,tTool\WObj:=wWobj;
        pTarget.trans:=[0*nScale,14.0*nScale,0];
        MoveL pTarget,vSpeed,z0,tTool\WObj:=wWobj;
        pTarget.trans:=[0*nScale,12.0*nScale,0];
        MoveL pTarget,vSpeed,z0,tTool\WObj:=wWobj;
        pTarget.trans:=[1*nScale,11.0*nScale,0];
        MoveL pTarget,vSpeed,z0,tTool\WObj:=wWobj;
        pTarget.trans:=[3*nScale,11.0*nScale,0];
        MoveL pTarget,vSpeed,z0,tTool\WObj:=wWobj;
        pTarget.trans:=[5*nScale,12.0*nScale,0];
        MoveL pTarget,vSpeed,z0,tTool\WObj:=wWobj;
        pTarget.trans:=[7*nScale,14.0*nScale,0];
        MoveL pTarget,vSpeed,z0,tTool\WObj:=wWobj;
        pTarget.trans:=[9*nScale,17.0*nScale,0];
        MoveL pTarget,vSpeed,fine,tTool\WObj:=wWobj;
        Reset do_pen;
        MoveL RelTool(pTarget,0,0,-2),vSpeed,z0,tTool\WObj:=wWobj;
        pTarget.trans:=[10*nScale,20.0*nScale,0];
        MoveL pTarget,vSpeed,fine,tTool\WObj:=wWobj;
        Set do_pen;
        pTarget.trans:=[4*nScale,2.0*nScale,0];
        MoveL pTarget,vSpeed,z0,tTool\WObj:=wWobj;
        pTarget.trans:=[3*nScale,0.0*nScale,0];
        MoveL pTarget,vSpeed,z0,tTool\WObj:=wWobj;
        pTarget.trans:=[1*nScale,-1.0*nScale,0];
        MoveL pTarget,vSpeed,z0,tTool\WObj:=wWobj;
        pTarget.trans:=[0*nScale,0.0*nScale,0];
        MoveL pTarget,vSpeed,z0,tTool\WObj:=wWobj;
        pTarget.trans:=[0*nScale,2.0*nScale,0];
        MoveL pTarget,vSpeed,z0,tTool\WObj:=wWobj;
        pTarget.trans:=[1*nScale,5.0*nScale,0];
        MoveL pTarget,vSpeed,z0,tTool\WObj:=wWobj;
        pTarget.trans:=[4*nScale,8.0*nScale,0];
        MoveL pTarget,vSpeed,z0,tTool\WObj:=wWobj;
        pTarget.trans:=[7*nScale,10.0*nScale,0];
        MoveL pTarget,vSpeed,z0,tTool\WObj:=wWobj;
        pTarget.trans:=[9*nScale,11.0*nScale,0];
        MoveL pTarget,vSpeed,z0,tTool\WObj:=wWobj;
        pTarget.trans:=[12*nScale,13.0*nScale,0];
        MoveL pTarget,vSpeed,z0,tTool\WObj:=wWobj;
        pTarget.trans:=[15*nScale,16.0*nScale,0];
        MoveL pTarget,vSpeed,fine,tTool\WObj:=wWobj;
        Reset do_pen;
        MoveL RelTool(pTarget,0,0,-2),vSpeed,z0,tTool\WObj:=wWobj;
        wWobj.oframe.trans.x:=wWobj.oframe.trans.x+15*nScale;
    ENDPROC

    ! Character: z
    PROC char_z(\num nScaleParam)
        VAR robtarget pTarget;
        VAR num nScale:=1;
        pTarget:=refTarget;
        IF Present(nScaleParam) THEN
            nScale:=nScaleParam;
        ENDIF
        pTarget.trans:=[0*nScale,16.0*nScale,0];
        MoveL pTarget,vSpeed,fine,tTool\WObj:=wWobj;
        Set do_pen;
        pTarget.trans:=[2*nScale,19.0*nScale,0];
        MoveL pTarget,vSpeed,z0,tTool\WObj:=wWobj;
        pTarget.trans:=[4*nScale,20.0*nScale,0];
        MoveL pTarget,vSpeed,z0,tTool\WObj:=wWobj;
        pTarget.trans:=[6*nScale,20.0*nScale,0];
        MoveL pTarget,vSpeed,z0,tTool\WObj:=wWobj;
        pTarget.trans:=[8*nScale,18.0*nScale,0];
        MoveL pTarget,vSpeed,z0,tTool\WObj:=wWobj;
        pTarget.trans:=[8*nScale,16.0*nScale,0];
        MoveL pTarget,vSpeed,z0,tTool\WObj:=wWobj;
        pTarget.trans:=[7*nScale,14.0*nScale,0];
        MoveL pTarget,vSpeed,z0,tTool\WObj:=wWobj;
        pTarget.trans:=[5*nScale,12.0*nScale,0];
        MoveL pTarget,vSpeed,z0,tTool\WObj:=wWobj;
        pTarget.trans:=[2*nScale,11.0*nScale,0];
        MoveL pTarget,vSpeed,z0,tTool\WObj:=wWobj;
        pTarget.trans:=[4*nScale,10.0*nScale,0];
        MoveL pTarget,vSpeed,z0,tTool\WObj:=wWobj;
        pTarget.trans:=[5*nScale,8.0*nScale,0];
        MoveL pTarget,vSpeed,z0,tTool\WObj:=wWobj;
        pTarget.trans:=[5*nScale,5.0*nScale,0];
        MoveL pTarget,vSpeed,z0,tTool\WObj:=wWobj;
        pTarget.trans:=[4*nScale,2.0*nScale,0];
        MoveL pTarget,vSpeed,z0,tTool\WObj:=wWobj;
        pTarget.trans:=[3*nScale,0.0*nScale,0];
        MoveL pTarget,vSpeed,z0,tTool\WObj:=wWobj;
        pTarget.trans:=[1*nScale,-1.0*nScale,0];
        MoveL pTarget,vSpeed,z0,tTool\WObj:=wWobj;
        pTarget.trans:=[0*nScale,0.0*nScale,0];
        MoveL pTarget,vSpeed,z0,tTool\WObj:=wWobj;
        pTarget.trans:=[0*nScale,2.0*nScale,0];
        MoveL pTarget,vSpeed,z0,tTool\WObj:=wWobj;
        pTarget.trans:=[1*nScale,5.0*nScale,0];
        MoveL pTarget,vSpeed,z0,tTool\WObj:=wWobj;
        pTarget.trans:=[4*nScale,8.0*nScale,0];
        MoveL pTarget,vSpeed,z0,tTool\WObj:=wWobj;
        pTarget.trans:=[7*nScale,10.0*nScale,0];
        MoveL pTarget,vSpeed,z0,tTool\WObj:=wWobj;
        pTarget.trans:=[11*nScale,13.0*nScale,0];
        MoveL pTarget,vSpeed,z0,tTool\WObj:=wWobj;
        pTarget.trans:=[14*nScale,16.0*nScale,0];
        MoveL pTarget,vSpeed,fine,tTool\WObj:=wWobj;
        Reset do_pen;
        MoveL RelTool(pTarget,0,0,-2),vSpeed,z0,tTool\WObj:=wWobj;
        wWobj.oframe.trans.x:=wWobj.oframe.trans.x+14*nScale;
    ENDPROC

    ! Character: A
    PROC char_upperA(\num nScaleParam)
        VAR robtarget pTarget;
        VAR num nScale:=1;
        pTarget:=refTarget;
        IF Present(nScaleParam) THEN
            nScale:=nScaleParam;
        ENDIF
        pTarget.trans:=[0*nScale,11.0*nScale,0];
        MoveL pTarget,vSpeed,fine,tTool\WObj:=wWobj;
        Set do_pen;
        pTarget.trans:=[2*nScale,12.0*nScale,0];
        MoveL pTarget,vSpeed,z0,tTool\WObj:=wWobj;
        pTarget.trans:=[5*nScale,15.0*nScale,0];
        MoveL pTarget,vSpeed,z0,tTool\WObj:=wWobj;
        pTarget.trans:=[8*nScale,19.0*nScale,0];
        MoveL pTarget,vSpeed,z0,tTool\WObj:=wWobj;
        pTarget.trans:=[12*nScale,26.0*nScale,0];
        MoveL pTarget,vSpeed,z0,tTool\WObj:=wWobj;
        pTarget.trans:=[15*nScale,32.0*nScale,0];
        MoveL pTarget,vSpeed,z0,tTool\WObj:=wWobj;
        pTarget.trans:=[15*nScale,11.0*nScale,0];
        MoveL pTarget,vSpeed,z0,tTool\WObj:=wWobj;
        pTarget.trans:=[14*nScale,14.0*nScale,0];
        MoveL pTarget,vSpeed,z0,tTool\WObj:=wWobj;
        pTarget.trans:=[12*nScale,17.0*nScale,0];
        MoveL pTarget,vSpeed,z0,tTool\WObj:=wWobj;
        pTarget.trans:=[10*nScale,19.0*nScale,0];
        MoveL pTarget,vSpeed,z0,tTool\WObj:=wWobj;
        pTarget.trans:=[7*nScale,21.0*nScale,0];
        MoveL pTarget,vSpeed,z0,tTool\WObj:=wWobj;
        pTarget.trans:=[5*nScale,21.0*nScale,0];
        MoveL pTarget,vSpeed,z0,tTool\WObj:=wWobj;
        pTarget.trans:=[4*nScale,20.0*nScale,0];
        MoveL pTarget,vSpeed,z0,tTool\WObj:=wWobj;
        pTarget.trans:=[4*nScale,18.0*nScale,0];
        MoveL pTarget,vSpeed,z0,tTool\WObj:=wWobj;
        pTarget.trans:=[5*nScale,16.0*nScale,0];
        MoveL pTarget,vSpeed,z0,tTool\WObj:=wWobj;
        pTarget.trans:=[7*nScale,14.0*nScale,0];
        MoveL pTarget,vSpeed,z0,tTool\WObj:=wWobj;
        pTarget.trans:=[10*nScale,12.0*nScale,0];
        MoveL pTarget,vSpeed,z0,tTool\WObj:=wWobj;
        pTarget.trans:=[13*nScale,11.0*nScale,0];
        MoveL pTarget,vSpeed,z0,tTool\WObj:=wWobj;
        pTarget.trans:=[18*nScale,11.0*nScale,0];
        MoveL pTarget,vSpeed,fine,tTool\WObj:=wWobj;
        Reset do_pen;
        MoveL RelTool(pTarget,0,0,-2),vSpeed,z0,tTool\WObj:=wWobj;
        wWobj.oframe.trans.x:=wWobj.oframe.trans.x+20*nScale;
    ENDPROC

    ! Character: B
    PROC char_upperB(\num nScaleParam)
        VAR robtarget pTarget;
        VAR num nScale:=1;
        pTarget:=refTarget;
        IF Present(nScaleParam) THEN
            nScale:=nScaleParam;
        ENDIF
        pTarget.trans:=[13*nScale,30.0*nScale,0];
        MoveL pTarget,vSpeed,fine,tTool\WObj:=wWobj;
        Set do_pen;
        pTarget.trans:=[14*nScale,29.0*nScale,0];
        MoveL pTarget,vSpeed,z0,tTool\WObj:=wWobj;
        pTarget.trans:=[14*nScale,26.0*nScale,0];
        MoveL pTarget,vSpeed,z0,tTool\WObj:=wWobj;
        pTarget.trans:=[13*nScale,22.0*nScale,0];
        MoveL pTarget,vSpeed,z0,tTool\WObj:=wWobj;
        pTarget.trans:=[12*nScale,19.0*nScale,0];
        MoveL pTarget,vSpeed,z0,tTool\WObj:=wWobj;
        pTarget.trans:=[11*nScale,17.0*nScale,0];
        MoveL pTarget,vSpeed,z0,tTool\WObj:=wWobj;
        pTarget.trans:=[9*nScale,14.0*nScale,0];
        MoveL pTarget,vSpeed,z0,tTool\WObj:=wWobj;
        pTarget.trans:=[7*nScale,12.0*nScale,0];
        MoveL pTarget,vSpeed,z0,tTool\WObj:=wWobj;
        pTarget.trans:=[5*nScale,11.0*nScale,0];
        MoveL pTarget,vSpeed,z0,tTool\WObj:=wWobj;
        pTarget.trans:=[4*nScale,11.0*nScale,0];
        MoveL pTarget,vSpeed,z0,tTool\WObj:=wWobj;
        pTarget.trans:=[3*nScale,12.0*nScale,0];
        MoveL pTarget,vSpeed,z0,tTool\WObj:=wWobj;
        pTarget.trans:=[3*nScale,15.0*nScale,0];
        MoveL pTarget,vSpeed,z0,tTool\WObj:=wWobj;
        pTarget.trans:=[4*nScale,20.0*nScale,0];
        MoveL pTarget,vSpeed,z0,tTool\WObj:=wWobj;
        pTarget.trans:=[5*nScale,23.0*nScale,0];
        MoveL pTarget,vSpeed,z0,tTool\WObj:=wWobj;
        pTarget.trans:=[6*nScale,25.0*nScale,0];
        MoveL pTarget,vSpeed,z0,tTool\WObj:=wWobj;
        pTarget.trans:=[8*nScale,28.0*nScale,0];
        MoveL pTarget,vSpeed,z0,tTool\WObj:=wWobj;
        pTarget.trans:=[10*nScale,30.0*nScale,0];
        MoveL pTarget,vSpeed,z0,tTool\WObj:=wWobj;
        pTarget.trans:=[12*nScale,31.0*nScale,0];
        MoveL pTarget,vSpeed,z0,tTool\WObj:=wWobj;
        pTarget.trans:=[15*nScale,32.0*nScale,0];
        MoveL pTarget,vSpeed,z0,tTool\WObj:=wWobj;
        pTarget.trans:=[18*nScale,32.0*nScale,0];
        MoveL pTarget,vSpeed,z0,tTool\WObj:=wWobj;
        pTarget.trans:=[20*nScale,31.0*nScale,0];
        MoveL pTarget,vSpeed,z0,tTool\WObj:=wWobj;
        pTarget.trans:=[21*nScale,29.0*nScale,0];
        MoveL pTarget,vSpeed,z0,tTool\WObj:=wWobj;
        pTarget.trans:=[21*nScale,27.0*nScale,0];
        MoveL pTarget,vSpeed,z0,tTool\WObj:=wWobj;
        pTarget.trans:=[20*nScale,25.0*nScale,0];
        MoveL pTarget,vSpeed,z0,tTool\WObj:=wWobj;
        pTarget.trans:=[19*nScale,24.0*nScale,0];
        MoveL pTarget,vSpeed,z0,tTool\WObj:=wWobj;
        pTarget.trans:=[17*nScale,23.0*nScale,0];
        MoveL pTarget,vSpeed,z0,tTool\WObj:=wWobj;
        pTarget.trans:=[14*nScale,22.0*nScale,0];
        MoveL pTarget,vSpeed,fine,tTool\WObj:=wWobj;
        Reset do_pen;
        MoveL RelTool(pTarget,0,0,-2),vSpeed,z0,tTool\WObj:=wWobj;
        pTarget.trans:=[13*nScale,22.0*nScale,0];
        MoveL pTarget,vSpeed,fine,tTool\WObj:=wWobj;
        Set do_pen;
        pTarget.trans:=[14*nScale,22.0*nScale,0];
        MoveL pTarget,vSpeed,z0,tTool\WObj:=wWobj;
        pTarget.trans:=[17*nScale,21.0*nScale,0];
        MoveL pTarget,vSpeed,z0,tTool\WObj:=wWobj;
        pTarget.trans:=[18*nScale,20.0*nScale,0];
        MoveL pTarget,vSpeed,z0,tTool\WObj:=wWobj;
        pTarget.trans:=[19*nScale,18.0*nScale,0];
        MoveL pTarget,vSpeed,z0,tTool\WObj:=wWobj;
        pTarget.trans:=[19*nScale,15.0*nScale,0];
        MoveL pTarget,vSpeed,z0,tTool\WObj:=wWobj;
        pTarget.trans:=[18*nScale,13.0*nScale,0];
        MoveL pTarget,vSpeed,z0,tTool\WObj:=wWobj;
        pTarget.trans:=[17*nScale,12.0*nScale,0];
        MoveL pTarget,vSpeed,z0,tTool\WObj:=wWobj;
        pTarget.trans:=[15*nScale,11.0*nScale,0];
        MoveL pTarget,vSpeed,z0,tTool\WObj:=wWobj;
        pTarget.trans:=[12*nScale,11.0*nScale,0];
        MoveL pTarget,vSpeed,z0,tTool\WObj:=wWobj;
        pTarget.trans:=[10*nScale,12.0*nScale,0];
        MoveL pTarget,vSpeed,z0,tTool\WObj:=wWobj;
        pTarget.trans:=[9*nScale,14.0*nScale,0];
        MoveL pTarget,vSpeed,fine,tTool\WObj:=wWobj;
        Reset do_pen;
        MoveL RelTool(pTarget,0,0,-2),vSpeed,z0,tTool\WObj:=wWobj;
        wWobj.oframe.trans.x:=wWobj.oframe.trans.x+23*nScale;
    ENDPROC

    ! Character: C
    PROC char_upperC(\num nScaleParam)
        VAR robtarget pTarget;
        VAR num nScale:=1;
        pTarget:=refTarget;
        IF Present(nScaleParam) THEN
            nScale:=nScaleParam;
        ENDIF
        pTarget.trans:=[12*nScale,26.0*nScale,0];
        MoveL pTarget,vSpeed,fine,tTool\WObj:=wWobj;
        Set do_pen;
        pTarget.trans:=[12*nScale,25.0*nScale,0];
        MoveL pTarget,vSpeed,z0,tTool\WObj:=wWobj;
        pTarget.trans:=[13*nScale,24.0*nScale,0];
        MoveL pTarget,vSpeed,z0,tTool\WObj:=wWobj;
        pTarget.trans:=[15*nScale,24.0*nScale,0];
        MoveL pTarget,vSpeed,z0,tTool\WObj:=wWobj;
        pTarget.trans:=[17*nScale,25.0*nScale,0];
        MoveL pTarget,vSpeed,z0,tTool\WObj:=wWobj;
        pTarget.trans:=[18*nScale,27.0*nScale,0];
        MoveL pTarget,vSpeed,z0,tTool\WObj:=wWobj;
        pTarget.trans:=[18*nScale,29.0*nScale,0];
        MoveL pTarget,vSpeed,z0,tTool\WObj:=wWobj;
        pTarget.trans:=[17*nScale,31.0*nScale,0];
        MoveL pTarget,vSpeed,z0,tTool\WObj:=wWobj;
        pTarget.trans:=[15*nScale,32.0*nScale,0];
        MoveL pTarget,vSpeed,z0,tTool\WObj:=wWobj;
        pTarget.trans:=[12*nScale,32.0*nScale,0];
        MoveL pTarget,vSpeed,z0,tTool\WObj:=wWobj;
        pTarget.trans:=[9*nScale,31.0*nScale,0];
        MoveL pTarget,vSpeed,z0,tTool\WObj:=wWobj;
        pTarget.trans:=[7*nScale,29.0*nScale,0];
        MoveL pTarget,vSpeed,z0,tTool\WObj:=wWobj;
        pTarget.trans:=[5*nScale,26.0*nScale,0];
        MoveL pTarget,vSpeed,z0,tTool\WObj:=wWobj;
        pTarget.trans:=[4*nScale,24.0*nScale,0];
        MoveL pTarget,vSpeed,z0,tTool\WObj:=wWobj;
        pTarget.trans:=[3*nScale,20.0*nScale,0];
        MoveL pTarget,vSpeed,z0,tTool\WObj:=wWobj;
        pTarget.trans:=[3*nScale,16.0*nScale,0];
        MoveL pTarget,vSpeed,z0,tTool\WObj:=wWobj;
        pTarget.trans:=[4*nScale,13.0*nScale,0];
        MoveL pTarget,vSpeed,z0,tTool\WObj:=wWobj;
        pTarget.trans:=[5*nScale,12.0*nScale,0];
        MoveL pTarget,vSpeed,z0,tTool\WObj:=wWobj;
        pTarget.trans:=[7*nScale,11.0*nScale,0];
        MoveL pTarget,vSpeed,z0,tTool\WObj:=wWobj;
        pTarget.trans:=[9*nScale,11.0*nScale,0];
        MoveL pTarget,vSpeed,z0,tTool\WObj:=wWobj;
        pTarget.trans:=[12*nScale,12.0*nScale,0];
        MoveL pTarget,vSpeed,z0,tTool\WObj:=wWobj;
        pTarget.trans:=[14*nScale,14.0*nScale,0];
        MoveL pTarget,vSpeed,z0,tTool\WObj:=wWobj;
        pTarget.trans:=[15*nScale,16.0*nScale,0];
        MoveL pTarget,vSpeed,fine,tTool\WObj:=wWobj;
        Reset do_pen;
        MoveL RelTool(pTarget,0,0,-2),vSpeed,z0,tTool\WObj:=wWobj;
        wWobj.oframe.trans.x:=wWobj.oframe.trans.x+20*nScale;
    ENDPROC

    ! Character: D
    PROC char_upperD(\num nScaleParam)
        VAR robtarget pTarget;
        VAR num nScale:=1;
        pTarget:=refTarget;
        IF Present(nScaleParam) THEN
            nScale:=nScaleParam;
        ENDIF
        pTarget.trans:=[13*nScale,32.0*nScale,0];
        MoveL pTarget,vSpeed,fine,tTool\WObj:=wWobj;
        Set do_pen;
        pTarget.trans:=[11*nScale,31.0*nScale,0];
        MoveL pTarget,vSpeed,z0,tTool\WObj:=wWobj;
        pTarget.trans:=[10*nScale,29.0*nScale,0];
        MoveL pTarget,vSpeed,z0,tTool\WObj:=wWobj;
        pTarget.trans:=[9*nScale,25.0*nScale,0];
        MoveL pTarget,vSpeed,z0,tTool\WObj:=wWobj;
        pTarget.trans:=[8*nScale,19.0*nScale,0];
        MoveL pTarget,vSpeed,z0,tTool\WObj:=wWobj;
        pTarget.trans:=[7*nScale,16.0*nScale,0];
        MoveL pTarget,vSpeed,z0,tTool\WObj:=wWobj;
        pTarget.trans:=[6*nScale,14.0*nScale,0];
        MoveL pTarget,vSpeed,z0,tTool\WObj:=wWobj;
        pTarget.trans:=[4*nScale,12.0*nScale,0];
        MoveL pTarget,vSpeed,z0,tTool\WObj:=wWobj;
        pTarget.trans:=[2*nScale,11.0*nScale,0];
        MoveL pTarget,vSpeed,z0,tTool\WObj:=wWobj;
        pTarget.trans:=[0*nScale,11.0*nScale,0];
        MoveL pTarget,vSpeed,z0,tTool\WObj:=wWobj;
        pTarget.trans:=[-1*nScale,12.0*nScale,0];
        MoveL pTarget,vSpeed,z0,tTool\WObj:=wWobj;
        pTarget.trans:=[-1*nScale,14.0*nScale,0];
        MoveL pTarget,vSpeed,z0,tTool\WObj:=wWobj;
        pTarget.trans:=[0*nScale,15.0*nScale,0];
        MoveL pTarget,vSpeed,z0,tTool\WObj:=wWobj;
        pTarget.trans:=[2*nScale,15.0*nScale,0];
        MoveL pTarget,vSpeed,z0,tTool\WObj:=wWobj;
        pTarget.trans:=[4*nScale,14.0*nScale,0];
        MoveL pTarget,vSpeed,z0,tTool\WObj:=wWobj;
        pTarget.trans:=[6*nScale,12.0*nScale,0];
        MoveL pTarget,vSpeed,z0,tTool\WObj:=wWobj;
        pTarget.trans:=[9*nScale,11.0*nScale,0];
        MoveL pTarget,vSpeed,z0,tTool\WObj:=wWobj;
        pTarget.trans:=[12*nScale,11.0*nScale,0];
        MoveL pTarget,vSpeed,z0,tTool\WObj:=wWobj;
        pTarget.trans:=[15*nScale,12.0*nScale,0];
        MoveL pTarget,vSpeed,z0,tTool\WObj:=wWobj;
        pTarget.trans:=[17*nScale,14.0*nScale,0];
        MoveL pTarget,vSpeed,z0,tTool\WObj:=wWobj;
        pTarget.trans:=[19*nScale,18.0*nScale,0];
        MoveL pTarget,vSpeed,z0,tTool\WObj:=wWobj;
        pTarget.trans:=[20*nScale,23.0*nScale,0];
        MoveL pTarget,vSpeed,z0,tTool\WObj:=wWobj;
        pTarget.trans:=[20*nScale,27.0*nScale,0];
        MoveL pTarget,vSpeed,z0,tTool\WObj:=wWobj;
        pTarget.trans:=[19*nScale,30.0*nScale,0];
        MoveL pTarget,vSpeed,z0,tTool\WObj:=wWobj;
        pTarget.trans:=[18*nScale,31.0*nScale,0];
        MoveL pTarget,vSpeed,z0,tTool\WObj:=wWobj;
        pTarget.trans:=[16*nScale,32.0*nScale,0];
        MoveL pTarget,vSpeed,z0,tTool\WObj:=wWobj;
        pTarget.trans:=[13*nScale,32.0*nScale,0];
        MoveL pTarget,vSpeed,z0,tTool\WObj:=wWobj;
        pTarget.trans:=[11*nScale,30.0*nScale,0];
        MoveL pTarget,vSpeed,z0,tTool\WObj:=wWobj;
        pTarget.trans:=[11*nScale,28.0*nScale,0];
        MoveL pTarget,vSpeed,z0,tTool\WObj:=wWobj;
        pTarget.trans:=[12*nScale,25.0*nScale,0];
        MoveL pTarget,vSpeed,z0,tTool\WObj:=wWobj;
        pTarget.trans:=[14*nScale,22.0*nScale,0];
        MoveL pTarget,vSpeed,z0,tTool\WObj:=wWobj;
        pTarget.trans:=[16*nScale,20.0*nScale,0];
        MoveL pTarget,vSpeed,z0,tTool\WObj:=wWobj;
        pTarget.trans:=[19*nScale,18.0*nScale,0];
        MoveL pTarget,vSpeed,z0,tTool\WObj:=wWobj;
        pTarget.trans:=[21*nScale,17.0*nScale,0];
        MoveL pTarget,vSpeed,fine,tTool\WObj:=wWobj;
        Reset do_pen;
        MoveL RelTool(pTarget,0,0,-2),vSpeed,z0,tTool\WObj:=wWobj;
        wWobj.oframe.trans.x:=wWobj.oframe.trans.x+23*nScale;
    ENDPROC

    ! Character: E
    PROC char_upperE(\num nScaleParam)
        VAR robtarget pTarget;
        VAR num nScale:=1;
        pTarget:=refTarget;
        IF Present(nScaleParam) THEN
            nScale:=nScaleParam;
        ENDIF
        pTarget.trans:=[14*nScale,28.0*nScale,0];
        MoveL pTarget,vSpeed,fine,tTool\WObj:=wWobj;
        Set do_pen;
        pTarget.trans:=[14*nScale,27.0*nScale,0];
        MoveL pTarget,vSpeed,z0,tTool\WObj:=wWobj;
        pTarget.trans:=[15*nScale,26.0*nScale,0];
        MoveL pTarget,vSpeed,z0,tTool\WObj:=wWobj;
        pTarget.trans:=[17*nScale,26.0*nScale,0];
        MoveL pTarget,vSpeed,z0,tTool\WObj:=wWobj;
        pTarget.trans:=[18*nScale,27.0*nScale,0];
        MoveL pTarget,vSpeed,z0,tTool\WObj:=wWobj;
        pTarget.trans:=[18*nScale,29.0*nScale,0];
        MoveL pTarget,vSpeed,z0,tTool\WObj:=wWobj;
        pTarget.trans:=[17*nScale,31.0*nScale,0];
        MoveL pTarget,vSpeed,z0,tTool\WObj:=wWobj;
        pTarget.trans:=[14*nScale,32.0*nScale,0];
        MoveL pTarget,vSpeed,z0,tTool\WObj:=wWobj;
        pTarget.trans:=[10*nScale,32.0*nScale,0];
        MoveL pTarget,vSpeed,z0,tTool\WObj:=wWobj;
        pTarget.trans:=[7*nScale,31.0*nScale,0];
        MoveL pTarget,vSpeed,z0,tTool\WObj:=wWobj;
        pTarget.trans:=[6*nScale,29.0*nScale,0];
        MoveL pTarget,vSpeed,z0,tTool\WObj:=wWobj;
        pTarget.trans:=[6*nScale,26.0*nScale,0];
        MoveL pTarget,vSpeed,z0,tTool\WObj:=wWobj;
        pTarget.trans:=[7*nScale,24.0*nScale,0];
        MoveL pTarget,vSpeed,z0,tTool\WObj:=wWobj;
        pTarget.trans:=[8*nScale,23.0*nScale,0];
        MoveL pTarget,vSpeed,z0,tTool\WObj:=wWobj;
        pTarget.trans:=[11*nScale,22.0*nScale,0];
        MoveL pTarget,vSpeed,z0,tTool\WObj:=wWobj;
        pTarget.trans:=[8*nScale,22.0*nScale,0];
        MoveL pTarget,vSpeed,z0,tTool\WObj:=wWobj;
        pTarget.trans:=[5*nScale,21.0*nScale,0];
        MoveL pTarget,vSpeed,z0,tTool\WObj:=wWobj;
        pTarget.trans:=[4*nScale,20.0*nScale,0];
        MoveL pTarget,vSpeed,z0,tTool\WObj:=wWobj;
        pTarget.trans:=[3*nScale,18.0*nScale,0];
        MoveL pTarget,vSpeed,z0,tTool\WObj:=wWobj;
        pTarget.trans:=[3*nScale,15.0*nScale,0];
        MoveL pTarget,vSpeed,z0,tTool\WObj:=wWobj;
        pTarget.trans:=[4*nScale,13.0*nScale,0];
        MoveL pTarget,vSpeed,z0,tTool\WObj:=wWobj;
        pTarget.trans:=[5*nScale,12.0*nScale,0];
        MoveL pTarget,vSpeed,z0,tTool\WObj:=wWobj;
        pTarget.trans:=[8*nScale,11.0*nScale,0];
        MoveL pTarget,vSpeed,z0,tTool\WObj:=wWobj;
        pTarget.trans:=[11*nScale,11.0*nScale,0];
        MoveL pTarget,vSpeed,z0,tTool\WObj:=wWobj;
        pTarget.trans:=[14*nScale,12.0*nScale,0];
        MoveL pTarget,vSpeed,z0,tTool\WObj:=wWobj;
        pTarget.trans:=[16*nScale,14.0*nScale,0];
        MoveL pTarget,vSpeed,z0,tTool\WObj:=wWobj;
        pTarget.trans:=[17*nScale,16.0*nScale,0];
        MoveL pTarget,vSpeed,fine,tTool\WObj:=wWobj;
        Reset do_pen;
        MoveL RelTool(pTarget,0,0,-2),vSpeed,z0,tTool\WObj:=wWobj;
        wWobj.oframe.trans.x:=wWobj.oframe.trans.x+20*nScale;
    ENDPROC

    ! Character: F
    PROC char_upperF(\num nScaleParam)
        VAR robtarget pTarget;
        VAR num nScale:=1;
        pTarget:=refTarget;
        IF Present(nScaleParam) THEN
            nScale:=nScaleParam;
        ENDIF
        pTarget.trans:=[10*nScale,26.0*nScale,0];
        MoveL pTarget,vSpeed,fine,tTool\WObj:=wWobj;
        Set do_pen;
        pTarget.trans:=[8*nScale,26.0*nScale,0];
        MoveL pTarget,vSpeed,z0,tTool\WObj:=wWobj;
        pTarget.trans:=[6*nScale,27.0*nScale,0];
        MoveL pTarget,vSpeed,z0,tTool\WObj:=wWobj;
        pTarget.trans:=[5*nScale,29.0*nScale,0];
        MoveL pTarget,vSpeed,z0,tTool\WObj:=wWobj;
        pTarget.trans:=[6*nScale,31.0*nScale,0];
        MoveL pTarget,vSpeed,z0,tTool\WObj:=wWobj;
        pTarget.trans:=[9*nScale,32.0*nScale,0];
        MoveL pTarget,vSpeed,z0,tTool\WObj:=wWobj;
        pTarget.trans:=[12*nScale,32.0*nScale,0];
        MoveL pTarget,vSpeed,z0,tTool\WObj:=wWobj;
        pTarget.trans:=[16*nScale,31.0*nScale,0];
        MoveL pTarget,vSpeed,z0,tTool\WObj:=wWobj;
        pTarget.trans:=[19*nScale,31.0*nScale,0];
        MoveL pTarget,vSpeed,z0,tTool\WObj:=wWobj;
        pTarget.trans:=[21*nScale,32.0*nScale,0];
        MoveL pTarget,vSpeed,fine,tTool\WObj:=wWobj;
        Reset do_pen;
        MoveL RelTool(pTarget,0,0,-2),vSpeed,z0,tTool\WObj:=wWobj;
        pTarget.trans:=[16*nScale,31.0*nScale,0];
        MoveL pTarget,vSpeed,fine,tTool\WObj:=wWobj;
        Set do_pen;
        pTarget.trans:=[14*nScale,24.0*nScale,0];
        MoveL pTarget,vSpeed,z0,tTool\WObj:=wWobj;
        pTarget.trans:=[12*nScale,18.0*nScale,0];
        MoveL pTarget,vSpeed,z0,tTool\WObj:=wWobj;
        pTarget.trans:=[10*nScale,14.0*nScale,0];
        MoveL pTarget,vSpeed,z0,tTool\WObj:=wWobj;
        pTarget.trans:=[8*nScale,12.0*nScale,0];
        MoveL pTarget,vSpeed,z0,tTool\WObj:=wWobj;
        pTarget.trans:=[6*nScale,11.0*nScale,0];
        MoveL pTarget,vSpeed,z0,tTool\WObj:=wWobj;
        pTarget.trans:=[4*nScale,11.0*nScale,0];
        MoveL pTarget,vSpeed,z0,tTool\WObj:=wWobj;
        pTarget.trans:=[2*nScale,12.0*nScale,0];
        MoveL pTarget,vSpeed,z0,tTool\WObj:=wWobj;
        pTarget.trans:=[1*nScale,14.0*nScale,0];
        MoveL pTarget,vSpeed,z0,tTool\WObj:=wWobj;
        pTarget.trans:=[1*nScale,16.0*nScale,0];
        MoveL pTarget,vSpeed,z0,tTool\WObj:=wWobj;
        pTarget.trans:=[2*nScale,17.0*nScale,0];
        MoveL pTarget,vSpeed,z0,tTool\WObj:=wWobj;
        pTarget.trans:=[4*nScale,17.0*nScale,0];
        MoveL pTarget,vSpeed,z0,tTool\WObj:=wWobj;
        pTarget.trans:=[6*nScale,16.0*nScale,0];
        MoveL pTarget,vSpeed,fine,tTool\WObj:=wWobj;
        Reset do_pen;
        MoveL RelTool(pTarget,0,0,-2),vSpeed,z0,tTool\WObj:=wWobj;
        pTarget.trans:=[9*nScale,22.0*nScale,0];
        MoveL pTarget,vSpeed,fine,tTool\WObj:=wWobj;
        Set do_pen;
        pTarget.trans:=[18*nScale,22.0*nScale,0];
        MoveL pTarget,vSpeed,fine,tTool\WObj:=wWobj;
        Reset do_pen;
        MoveL RelTool(pTarget,0,0,-2),vSpeed,z0,tTool\WObj:=wWobj;
        wWobj.oframe.trans.x:=wWobj.oframe.trans.x+20*nScale;
    ENDPROC

    ! Character: G
    PROC char_upperG(\num nScaleParam)
        VAR robtarget pTarget;
        VAR num nScale:=1;
        pTarget:=refTarget;
        IF Present(nScaleParam) THEN
            nScale:=nScaleParam;
        ENDIF
        pTarget.trans:=[0*nScale,11.0*nScale,0];
        MoveL pTarget,vSpeed,fine,tTool\WObj:=wWobj;
        Set do_pen;
        pTarget.trans:=[2*nScale,12.0*nScale,0];
        MoveL pTarget,vSpeed,z0,tTool\WObj:=wWobj;
        pTarget.trans:=[6*nScale,16.0*nScale,0];
        MoveL pTarget,vSpeed,z0,tTool\WObj:=wWobj;
        pTarget.trans:=[9*nScale,21.0*nScale,0];
        MoveL pTarget,vSpeed,z0,tTool\WObj:=wWobj;
        pTarget.trans:=[10*nScale,24.0*nScale,0];
        MoveL pTarget,vSpeed,z0,tTool\WObj:=wWobj;
        pTarget.trans:=[11*nScale,28.0*nScale,0];
        MoveL pTarget,vSpeed,z0,tTool\WObj:=wWobj;
        pTarget.trans:=[11*nScale,31.0*nScale,0];
        MoveL pTarget,vSpeed,z0,tTool\WObj:=wWobj;
        pTarget.trans:=[10*nScale,32.0*nScale,0];
        MoveL pTarget,vSpeed,z0,tTool\WObj:=wWobj;
        pTarget.trans:=[9*nScale,32.0*nScale,0];
        MoveL pTarget,vSpeed,z0,tTool\WObj:=wWobj;
        pTarget.trans:=[8*nScale,31.0*nScale,0];
        MoveL pTarget,vSpeed,z0,tTool\WObj:=wWobj;
        pTarget.trans:=[7*nScale,29.0*nScale,0];
        MoveL pTarget,vSpeed,z0,tTool\WObj:=wWobj;
        pTarget.trans:=[7*nScale,26.0*nScale,0];
        MoveL pTarget,vSpeed,z0,tTool\WObj:=wWobj;
        pTarget.trans:=[8*nScale,24.0*nScale,0];
        MoveL pTarget,vSpeed,z0,tTool\WObj:=wWobj;
        pTarget.trans:=[10*nScale,23.0*nScale,0];
        MoveL pTarget,vSpeed,z0,tTool\WObj:=wWobj;
        pTarget.trans:=[14*nScale,23.0*nScale,0];
        MoveL pTarget,vSpeed,z0,tTool\WObj:=wWobj;
        pTarget.trans:=[17*nScale,24.0*nScale,0];
        MoveL pTarget,vSpeed,z0,tTool\WObj:=wWobj;
        pTarget.trans:=[18*nScale,25.0*nScale,0];
        MoveL pTarget,vSpeed,z0,tTool\WObj:=wWobj;
        pTarget.trans:=[19*nScale,27.0*nScale,0];
        MoveL pTarget,vSpeed,z0,tTool\WObj:=wWobj;
        pTarget.trans:=[19*nScale,21.0*nScale,0];
        MoveL pTarget,vSpeed,z0,tTool\WObj:=wWobj;
        pTarget.trans:=[18*nScale,16.0*nScale,0];
        MoveL pTarget,vSpeed,z0,tTool\WObj:=wWobj;
        pTarget.trans:=[17*nScale,14.0*nScale,0];
        MoveL pTarget,vSpeed,z0,tTool\WObj:=wWobj;
        pTarget.trans:=[15*nScale,12.0*nScale,0];
        MoveL pTarget,vSpeed,z0,tTool\WObj:=wWobj;
        pTarget.trans:=[12*nScale,11.0*nScale,0];
        MoveL pTarget,vSpeed,z0,tTool\WObj:=wWobj;
        pTarget.trans:=[8*nScale,11.0*nScale,0];
        MoveL pTarget,vSpeed,z0,tTool\WObj:=wWobj;
        pTarget.trans:=[5*nScale,12.0*nScale,0];
        MoveL pTarget,vSpeed,z0,tTool\WObj:=wWobj;
        pTarget.trans:=[3*nScale,14.0*nScale,0];
        MoveL pTarget,vSpeed,z0,tTool\WObj:=wWobj;
        pTarget.trans:=[2*nScale,16.0*nScale,0];
        MoveL pTarget,vSpeed,z0,tTool\WObj:=wWobj;
        pTarget.trans:=[2*nScale,18.0*nScale,0];
        MoveL pTarget,vSpeed,fine,tTool\WObj:=wWobj;
        Reset do_pen;
        MoveL RelTool(pTarget,0,0,-2),vSpeed,z0,tTool\WObj:=wWobj;
        wWobj.oframe.trans.x:=wWobj.oframe.trans.x+23*nScale;
    ENDPROC

    ! Character: H
    PROC char_upperH(\num nScaleParam)
        VAR robtarget pTarget;
        VAR num nScale:=1;
        pTarget:=refTarget;
        IF Present(nScaleParam) THEN
            nScale:=nScaleParam;
        ENDIF
        pTarget.trans:=[7*nScale,25.0*nScale,0];
        MoveL pTarget,vSpeed,fine,tTool\WObj:=wWobj;
        Set do_pen;
        pTarget.trans:=[5*nScale,26.0*nScale,0];
        MoveL pTarget,vSpeed,z0,tTool\WObj:=wWobj;
        pTarget.trans:=[4*nScale,28.0*nScale,0];
        MoveL pTarget,vSpeed,z0,tTool\WObj:=wWobj;
        pTarget.trans:=[4*nScale,29.0*nScale,0];
        MoveL pTarget,vSpeed,z0,tTool\WObj:=wWobj;
        pTarget.trans:=[5*nScale,31.0*nScale,0];
        MoveL pTarget,vSpeed,z0,tTool\WObj:=wWobj;
        pTarget.trans:=[7*nScale,32.0*nScale,0];
        MoveL pTarget,vSpeed,z0,tTool\WObj:=wWobj;
        pTarget.trans:=[8*nScale,32.0*nScale,0];
        MoveL pTarget,vSpeed,z0,tTool\WObj:=wWobj;
        pTarget.trans:=[10*nScale,31.0*nScale,0];
        MoveL pTarget,vSpeed,z0,tTool\WObj:=wWobj;
        pTarget.trans:=[11*nScale,29.0*nScale,0];
        MoveL pTarget,vSpeed,z0,tTool\WObj:=wWobj;
        pTarget.trans:=[11*nScale,27.0*nScale,0];
        MoveL pTarget,vSpeed,z0,tTool\WObj:=wWobj;
        pTarget.trans:=[10*nScale,23.0*nScale,0];
        MoveL pTarget,vSpeed,z0,tTool\WObj:=wWobj;
        pTarget.trans:=[8*nScale,17.0*nScale,0];
        MoveL pTarget,vSpeed,z0,tTool\WObj:=wWobj;
        pTarget.trans:=[6*nScale,13.0*nScale,0];
        MoveL pTarget,vSpeed,z0,tTool\WObj:=wWobj;
        pTarget.trans:=[4*nScale,11.0*nScale,0];
        MoveL pTarget,vSpeed,z0,tTool\WObj:=wWobj;
        pTarget.trans:=[2*nScale,11.0*nScale,0];
        MoveL pTarget,vSpeed,z0,tTool\WObj:=wWobj;
        pTarget.trans:=[1*nScale,12.0*nScale,0];
        MoveL pTarget,vSpeed,z0,tTool\WObj:=wWobj;
        pTarget.trans:=[1*nScale,14.0*nScale,0];
        MoveL pTarget,vSpeed,fine,tTool\WObj:=wWobj;
        Reset do_pen;
        MoveL RelTool(pTarget,0,0,-2),vSpeed,z0,tTool\WObj:=wWobj;
        pTarget.trans:=[7*nScale,20.0*nScale,0];
        MoveL pTarget,vSpeed,fine,tTool\WObj:=wWobj;
        Set do_pen;
        pTarget.trans:=[16*nScale,23.0*nScale,0];
        MoveL pTarget,vSpeed,z0,tTool\WObj:=wWobj;
        pTarget.trans:=[18*nScale,24.0*nScale,0];
        MoveL pTarget,vSpeed,z0,tTool\WObj:=wWobj;
        pTarget.trans:=[21*nScale,26.0*nScale,0];
        MoveL pTarget,vSpeed,z0,tTool\WObj:=wWobj;
        pTarget.trans:=[23*nScale,28.0*nScale,0];
        MoveL pTarget,vSpeed,z0,tTool\WObj:=wWobj;
        pTarget.trans:=[24*nScale,30.0*nScale,0];
        MoveL pTarget,vSpeed,z0,tTool\WObj:=wWobj;
        pTarget.trans:=[24*nScale,31.0*nScale,0];
        MoveL pTarget,vSpeed,z0,tTool\WObj:=wWobj;
        pTarget.trans:=[23*nScale,32.0*nScale,0];
        MoveL pTarget,vSpeed,z0,tTool\WObj:=wWobj;
        pTarget.trans:=[22*nScale,32.0*nScale,0];
        MoveL pTarget,vSpeed,z0,tTool\WObj:=wWobj;
        pTarget.trans:=[20*nScale,30.0*nScale,0];
        MoveL pTarget,vSpeed,z0,tTool\WObj:=wWobj;
        pTarget.trans:=[18*nScale,26.0*nScale,0];
        MoveL pTarget,vSpeed,z0,tTool\WObj:=wWobj;
        pTarget.trans:=[16*nScale,20.0*nScale,0];
        MoveL pTarget,vSpeed,z0,tTool\WObj:=wWobj;
        pTarget.trans:=[15*nScale,15.0*nScale,0];
        MoveL pTarget,vSpeed,z0,tTool\WObj:=wWobj;
        pTarget.trans:=[15*nScale,12.0*nScale,0];
        MoveL pTarget,vSpeed,z0,tTool\WObj:=wWobj;
        pTarget.trans:=[16*nScale,11.0*nScale,0];
        MoveL pTarget,vSpeed,z0,tTool\WObj:=wWobj;
        pTarget.trans:=[17*nScale,11.0*nScale,0];
        MoveL pTarget,vSpeed,z0,tTool\WObj:=wWobj;
        pTarget.trans:=[19*nScale,12.0*nScale,0];
        MoveL pTarget,vSpeed,z0,tTool\WObj:=wWobj;
        pTarget.trans:=[20*nScale,13.0*nScale,0];
        MoveL pTarget,vSpeed,z0,tTool\WObj:=wWobj;
        pTarget.trans:=[22*nScale,16.0*nScale,0];
        MoveL pTarget,vSpeed,fine,tTool\WObj:=wWobj;
        Reset do_pen;
        MoveL RelTool(pTarget,0,0,-2),vSpeed,z0,tTool\WObj:=wWobj;
        wWobj.oframe.trans.x:=wWobj.oframe.trans.x+24*nScale;
    ENDPROC

